LIN {X 0,Y 586.266,Z 608.093,A -85,B 0,C 180,E1 26221.406,E2 26221.406} C_VEL
LIN {X 0,Y 585.812,Z 650.287,A -85,B 0,C 180,E1 26218.326,E2 26218.326} C_VEL
LIN {X 0,Y 585.394,Z 696.233,A -85,B 0,C 180,E1 26215.061,E2 26215.061} C_VEL
LIN {X 0,Y 585.368,Z 709.809,A -85,B 0,C 180,E1 26214.141,E2 26214.141} C_VEL
LIN {X 0,Y 585.877,Z 715.244,A -85,B 0,C 180,E1 26214.043,E2 26214.043} C_VEL
LIN {X 0,Y 585.444,Z 927.531,A -85,B 0,C 180,E1 26211.27,E2 26211.27} C_VEL
LIN {X 0,Y 585.33,Z 946.86,A -85,B 0,C 180,E1 26210.828,E2 26210.828} C_VEL
LIN {X 0,Y 585.19,Z 964.794,A -85,B 0,C 180,E1 26210.242,E2 26210.242} C_VEL
LIN {X 0,Y 585.02,Z 982.786,A -85,B 0,C 180,E1 26209.467,E2 26209.467} C_VEL
LIN {X 0,Y 584.825,Z 1000.721,A -85,B 0,C 180,E1 26208.49,E2 26208.49} C_VEL
LIN {X 0,Y 584.635,Z 1017.158,A -85,B 0,C 180,E1 26207.388,E2 26207.388} C_VEL
LIN {X 0,Y 584.458,Z 1032.33,A -85,B 0,C 180,E1 26206.161,E2 26206.161} C_VEL
LIN {X 0,Y 584.295,Z 1046.685,A -85,B 0,C 180,E1 26204.772,E2 26204.772} C_VEL
LIN {X 0,Y 584.162,Z 1059.749,A -85,B 0,C 180,E1 26203.259,E2 26203.259} C_VEL
LIN {X 0,Y 584.061,Z 1071.294,A -85,B 0,C 180,E1 26201.654,E2 26201.654} C_VEL
LIN {X 0,Y 583.991,Z 1081.331,A -85,B 0,C 180,E1 26199.958,E2 26199.958} C_VEL
LIN {X 0,Y 583.953,Z 1089.534,A -85,B 0,C 180,E1 26198.244,E2 26198.244} C_VEL
LIN {X 0,Y 583.927,Z 1096.129,A -85,B 0,C 180,E1 26196.489,E2 26196.489} C_VEL
LIN {X 0,Y 583.916,Z 1101.299,A -85,B 0,C 180,E1 26194.616,E2 26194.616} C_VEL
LIN {X 0,Y 583.904,Z 1104.662,A -85,B 0,C 180,E1 26192.748,E2 26192.748} C_VEL
LIN {X 0,Y 583.911,Z 1106.306,A -85,B 0,C 180,E1 26190.883,E2 26190.883} C_VEL
LIN {X 0,Y 583.908,Z 1106.262,A -85,B 0,C 180,E1 26189.019,E2 26189.019} C_VEL
LIN {X 0,Y 583.906,Z 1104.537,A -85,B 0,C 180,E1 26187.153,E2 26187.153} C_VEL
LIN {X 0,Y 583.919,Z 1101.014,A -85,B 0,C 180,E1 26185.255,E2 26185.255} C_VEL
LIN {X 0,Y 583.926,Z 1095.819,A -85,B 0,C 180,E1 26183.412,E2 26183.412} C_VEL
LIN {X 0,Y 583.963,Z 1088.595,A -85,B 0,C 180,E1 26181.532,E2 26181.532} C_VEL
LIN {X 0,Y 584.009,Z 1079.736,A -85,B 0,C 180,E1 26179.743,E2 26179.743} C_VEL
LIN {X 0,Y 584.082,Z 1069.314,A -85,B 0,C 180,E1 26178.045,E2 26178.045} C_VEL
LIN {X 0,Y 584.186,Z 1057.326,A -85,B 0,C 180,E1 26176.439,E2 26176.439} C_VEL
LIN {X 0,Y 584.319,Z 1044.137,A -85,B 0,C 180,E1 26174.965,E2 26174.965} C_VEL
LIN {X 0,Y 584.478,Z 1029.579,A -85,B 0,C 180,E1 26173.604,E2 26173.604} C_VEL
LIN {X 0,Y 584.658,Z 1013.886,A -85,B 0,C 180,E1 26172.38,E2 26172.38} C_VEL
LIN {X 0,Y 584.848,Z 996.836,A -85,B 0,C 180,E1 26171.284,E2 26171.284} C_VEL
LIN {X 0,Y 585.039,Z 978.544,A -85,B 0,C 180,E1 26170.336,E2 26170.336} C_VEL
LIN {X 0,Y 585.211,Z 960.378,A -85,B 0,C 180,E1 26169.601,E2 26169.601} C_VEL
LIN {X 0,Y 585.358,Z 940.959,A -85,B 0,C 180,E1 26169.021,E2 26169.021} C_VEL
LIN {X 0,Y 585.468,Z 921.478,A -85,B 0,C 180,E1 26168.636,E2 26168.636} C_VEL
LIN {X 0,Y 585.728,Z 711.988,A -85,B 0,C 180,E1 26165.908,E2 26165.908} C_VEL
LIN {X 0,Y 585.285,Z 708.498,A -85,B 0,C 180,E1 26165.795,E2 26165.795} C_VEL
LIN {X 0,Y 585.682,Z 666.013,A -85,B 0,C 180,E1 26162.802,E2 26162.802} C_VEL
LIN {X 0,Y 586.142,Z 620.088,A -85,B 0,C 180,E1 26159.479,E2 26159.479} C_VEL
LIN {X 0,Y 586.104,Z 607.396,A -85,B 0,C 180,E1 26158.532,E2 26158.532} C_VEL
LIN {X 0,Y 584.094,Z 601.706,A -85,B 0,C 180,E1 26157.949,E2 26157.949} C_VEL
LIN {X 0,Y 584.092,Z 601.478,A -85,B 0,C 180,E1 26154.888,E2 26154.888} C_VEL
LIN {X 0,Y 584.068,Z 601.478,A -85,B 0,C 180,E1 26151.705,E2 26151.705} C_VEL
LIN {X 0,Y 584.088,Z 601.475,A -85,B 0,C 180,E1 26148.51,E2 26148.51} C_VEL
LIN {X 0,Y 584.079,Z 601.478,A -85,B 0,C 180,E1 26145.269,E2 26145.269} C_VEL
LIN {X 0,Y 584.092,Z 601.472,A -85,B 0,C 180,E1 26142.015,E2 26142.015} C_VEL
LIN {X 0,Y 584.093,Z 601.481,A -85,B 0,C 180,E1 26138.668,E2 26138.668} C_VEL
LIN {X 0,Y 584.089,Z 601.473,A -85,B 0,C 180,E1 26135.352,E2 26135.352} C_VEL
LIN {X 0,Y 584.073,Z 601.478,A -85,B 0,C 180,E1 26132.167,E2 26132.167} C_VEL
LIN {X 0,Y 584.091,Z 601.475,A -85,B 0,C 180,E1 26128.976,E2 26128.976} C_VEL
LIN {X 0,Y 584.063,Z 601.477,A -85,B 0,C 180,E1 26125.774,E2 26125.774} C_VEL
LIN {X 0,Y 584.096,Z 601.479,A -85,B 0,C 180,E1 26122.547,E2 26122.547} C_VEL
LIN {X 0,Y 584.058,Z 601.476,A -85,B 0,C 180,E1 26119.391,E2 26119.391} C_VEL
LIN {X 0,Y 584.09,Z 601.482,A -85,B 0,C 180,E1 26116.1,E2 26116.1} C_VEL
LIN {X 0,Y 584.06,Z 601.476,A -85,B 0,C 180,E1 26112.959,E2 26112.959} C_VEL
LIN {X 0,Y 584.053,Z 601.481,A -85,B 0,C 180,E1 26109.558,E2 26109.558} C_VEL
LIN {X 0,Y 584.073,Z 601.479,A -85,B 0,C 180,E1 26106.487,E2 26106.487} C_VEL
LIN {X 0,Y 584.084,Z 601.735,A -85,B 0,C 180,E1 26104.652,E2 26104.652} C_VEL
LIN {X 0,Y 584.958,Z 606.283,A -85,B 0,C 180,E1 26104.117,E2 26104.117} C_VEL
LIN {X 0,Y 584.765,Z 632.877,A -85,B 0,C 180,E1 26101.078,E2 26101.078} C_VEL
LIN {X 0,Y 584.541,Z 663.315,A -85,B 0,C 180,E1 26097.647,E2 26097.647} C_VEL
LIN {X 0,Y 584.373,Z 692.632,A -85,B 0,C 180,E1 26094.428,E2 26094.428} C_VEL
LIN {X 0,Y 584.842,Z 698.032,A -85,B 0,C 180,E1 26094.331,E2 26094.331} C_VEL
LIN {X 0,Y 584.731,Z 757.317,A -85,B 0,C 180,E1 26093.592,E2 26093.592} C_VEL
LIN {X 0,Y 583.768,Z 764.99,A -85,B 0,C 180,E1 26093.522,E2 26093.522} C_VEL
LIN {X 0,Y 577.692,Z 785.335,A -85,B 0,C 180,E1 26093.433,E2 26093.433} C_VEL
LIN {X 0,Y 576.962,Z 791.923,A -85,B 0,C 180,E1 26093.37,E2 26093.37} C_VEL
LIN {X 0,Y 576.9,Z 833.418,A -85,B 0,C 180,E1 26092.816,E2 26092.816} C_VEL
LIN {X 0,Y 576.808,Z 850.257,A -85,B 0,C 180,E1 26092.395,E2 26092.395} C_VEL
LIN {X 0,Y 576.673,Z 865.421,A -85,B 0,C 180,E1 26091.826,E2 26091.826} C_VEL
LIN {X 0,Y 576.524,Z 880.375,A -85,B 0,C 180,E1 26091.07,E2 26091.07} C_VEL
LIN {X 0,Y 576.387,Z 894.173,A -85,B 0,C 180,E1 26090.169,E2 26090.169} C_VEL
LIN {X 0,Y 576.244,Z 907.214,A -85,B 0,C 180,E1 26089.098,E2 26089.098} C_VEL
LIN {X 0,Y 576.128,Z 919.088,A -85,B 0,C 180,E1 26087.878,E2 26087.878} C_VEL
LIN {X 0,Y 576.036,Z 929.428,A -85,B 0,C 180,E1 26086.55,E2 26086.55} C_VEL
LIN {X 0,Y 575.976,Z 938.273,A -85,B 0,C 180,E1 26085.112,E2 26085.112} C_VEL
LIN {X 0,Y 575.94,Z 945.143,A -85,B 0,C 180,E1 26083.666,E2 26083.666} C_VEL
LIN {X 0,Y 575.921,Z 950.718,A -85,B 0,C 180,E1 26082.062,E2 26082.062} C_VEL
LIN {X 0,Y 575.916,Z 954.279,A -85,B 0,C 180,E1 26080.513,E2 26080.513} C_VEL
LIN {X 0,Y 575.913,Z 956.237,A -85,B 0,C 180,E1 26078.797,E2 26078.797} C_VEL
LIN {X 0,Y 575.915,Z 956.297,A -85,B 0,C 180,E1 26077.204,E2 26077.204} C_VEL
LIN {X 0,Y 575.916,Z 954.417,A -85,B 0,C 180,E1 26075.485,E2 26075.485} C_VEL
LIN {X 0,Y 575.921,Z 951.002,A -85,B 0,C 180,E1 26073.945,E2 26073.945} C_VEL
LIN {X 0,Y 575.937,Z 945.71,A -85,B 0,C 180,E1 26072.385,E2 26072.385} C_VEL
LIN {X 0,Y 575.972,Z 938.918,A -85,B 0,C 180,E1 26070.917,E2 26070.917} C_VEL
LIN {X 0,Y 576.033,Z 929.921,A -85,B 0,C 180,E1 26069.43,E2 26069.43} C_VEL
LIN {X 0,Y 576.127,Z 919.385,A -85,B 0,C 180,E1 26068.066,E2 26068.066} C_VEL
LIN {X 0,Y 576.239,Z 907.818,A -85,B 0,C 180,E1 26066.868,E2 26066.868} C_VEL
LIN {X 0,Y 576.376,Z 895.002,A -85,B 0,C 180,E1 26065.802,E2 26065.802} C_VEL
LIN {X 0,Y 576.518,Z 881.624,A -85,B 0,C 180,E1 26064.912,E2 26064.912} C_VEL
LIN {X 0,Y 576.662,Z 866.294,A -85,B 0,C 180,E1 26064.122,E2 26064.122} C_VEL
LIN {X 0,Y 576.807,Z 850.362,A -85,B 0,C 180,E1 26063.518,E2 26063.518} C_VEL
LIN {X 0,Y 576.897,Z 833.646,A -85,B 0,C 180,E1 26063.099,E2 26063.099} C_VEL
LIN {X 0,Y 576.958,Z 794.896,A -85,B 0,C 180,E1 26062.578,E2 26062.578} C_VEL
LIN {X 0,Y 576.936,Z 695.316,A -85,B 0,C 180,E1 26061.314,E2 26061.314} C_VEL
LIN {X 0,Y 576.519,Z 692.432,A -85,B 0,C 180,E1 26061.238,E2 26061.238} C_VEL
LIN {X 0,Y 576.769,Z 663.417,A -85,B 0,C 180,E1 26057.998,E2 26057.998} C_VEL
LIN {X 0,Y 577.081,Z 633.4,A -85,B 0,C 180,E1 26054.565,E2 26054.565} C_VEL
LIN {X 0,Y 577.283,Z 607.484,A -85,B 0,C 180,E1 26051.59,E2 26051.59} C_VEL
LIN {X 0,Y 576.093,Z 602.542,A -85,B 0,C 180,E1 26050.936,E2 26050.936} C_VEL
LIN {X 0,Y 576.161,Z 602.456,A -85,B 0,C 180,E1 26047.777,E2 26047.777} C_VEL
LIN {X 0,Y 576.088,Z 602.47,A -85,B 0,C 180,E1 26044.646,E2 26044.646} C_VEL
LIN {X 0,Y 576.163,Z 602.467,A -85,B 0,C 180,E1 26041.49,E2 26041.49} C_VEL
LIN {X 0,Y 576.094,Z 602.468,A -85,B 0,C 180,E1 26038.364,E2 26038.364} C_VEL
LIN {X 0,Y 576.159,Z 602.459,A -85,B 0,C 180,E1 26035.162,E2 26035.162} C_VEL
LIN {X 0,Y 576.1,Z 602.469,A -85,B 0,C 180,E1 26032.017,E2 26032.017} C_VEL
LIN {X 0,Y 576.154,Z 602.466,A -85,B 0,C 180,E1 26028.832,E2 26028.832} C_VEL
LIN {X 0,Y 576.106,Z 602.465,A -85,B 0,C 180,E1 26025.709,E2 26025.709} C_VEL
LIN {X 0,Y 576.145,Z 602.467,A -85,B 0,C 180,E1 26022.427,E2 26022.427} C_VEL
LIN {X 0,Y 576.16,Z 602.725,A -85,B 0,C 180,E1 26020.108,E2 26020.108} C_VEL
LIN {X 0,Y 577.539,Z 609.023,A -85,B 0,C 180,E1 26019.266,E2 26019.266} C_VEL
LIN {X 0,Y 577.051,Z 635.9,A -85,B 0,C 180,E1 26016.067,E2 26016.067} C_VEL
LIN {X 0,Y 576.75,Z 663.687,A -85,B 0,C 180,E1 26012.882,E2 26012.882} C_VEL
LIN {X 0,Y 576.515,Z 692.398,A -85,B 0,C 180,E1 26009.677,E2 26009.677} C_VEL
LIN {X 0,Y 577.137,Z 698.434,A -85,B 0,C 180,E1 26009.55,E2 26009.55} C_VEL
LIN {X 0,Y 576.9,Z 832.64,A -85,B 0,C 180,E1 26007.831,E2 26007.831} C_VEL
LIN {X 0,Y 576.81,Z 849.612,A -85,B 0,C 180,E1 26007.414,E2 26007.414} C_VEL
LIN {X 0,Y 576.689,Z 864.449,A -85,B 0,C 180,E1 26006.87,E2 26006.87} C_VEL
LIN {X 0,Y 576.537,Z 879.449,A -85,B 0,C 180,E1 26006.122,E2 26006.122} C_VEL
LIN {X 0,Y 576.396,Z 893.447,A -85,B 0,C 180,E1 26005.224,E2 26005.224} C_VEL
LIN {X 0,Y 576.254,Z 906.354,A -85,B 0,C 180,E1 26004.175,E2 26004.175} C_VEL
LIN {X 0,Y 576.139,Z 917.811,A -85,B 0,C 180,E1 26003.023,E2 26003.023} C_VEL
LIN {X 0,Y 576.047,Z 928.241,A -85,B 0,C 180,E1 26001.717,E2 26001.717} C_VEL
LIN {X 0,Y 575.98,Z 937.191,A -85,B 0,C 180,E1 26000.306,E2 26000.306} C_VEL
LIN {X 0,Y 575.944,Z 944.215,A -85,B 0,C 180,E1 25998.89,E2 25998.89} C_VEL
LIN {X 0,Y 575.926,Z 949.881,A -85,B 0,C 180,E1 25997.34,E2 25997.34} C_VEL
LIN {X 0,Y 575.916,Z 953.885,A -85,B 0,C 180,E1 25995.728,E2 25995.728} C_VEL
LIN {X 0,Y 575.914,Z 956.024,A -85,B 0,C 180,E1 25994.116,E2 25994.116} C_VEL
LIN {X 0,Y 575.915,Z 956.385,A -85,B 0,C 180,E1 25992.417,E2 25992.417} C_VEL
LIN {X 0,Y 575.917,Z 954.935,A -85,B 0,C 180,E1 25990.813,E2 25990.813} C_VEL
LIN {X 0,Y 575.923,Z 951.544,A -85,B 0,C 180,E1 25989.152,E2 25989.152} C_VEL
LIN {X 0,Y 575.936,Z 946.78,A -85,B 0,C 180,E1 25987.654,E2 25987.654} C_VEL
LIN {X 0,Y 575.963,Z 940.059,A -85,B 0,C 180,E1 25986.142,E2 25986.142} C_VEL
LIN {X 0,Y 576.021,Z 931.862,A -85,B 0,C 180,E1 25984.722,E2 25984.722} C_VEL
LIN {X 0,Y 576.098,Z 922.181,A -85,B 0,C 180,E1 25983.399,E2 25983.399} C_VEL
LIN {X 0,Y 576.214,Z 910.366,A -85,B 0,C 180,E1 25982.111,E2 25982.111} C_VEL
LIN {X 0,Y 576.342,Z 898.277,A -85,B 0,C 180,E1 25981.052,E2 25981.052} C_VEL
LIN {X 0,Y 576.483,Z 884.619,A -85,B 0,C 180,E1 25980.096,E2 25980.096} C_VEL
LIN {X 0,Y 576.628,Z 870.151,A -85,B 0,C 180,E1 25979.298,E2 25979.298} C_VEL
LIN {X 0,Y 576.765,Z 854.672,A -85,B 0,C 180,E1 25978.663,E2 25978.663} C_VEL
LIN {X 0,Y 576.881,Z 838.179,A -85,B 0,C 180,E1 25978.19,E2 25978.19} C_VEL
LIN {X 0,Y 576.944,Z 820.063,A -85,B 0,C 180,E1 25977.895,E2 25977.895} C_VEL
LIN {X 0,Y 576.927,Z 695.244,A -85,B 0,C 180,E1 25976.313,E2 25976.313} C_VEL
LIN {X 0,Y 576.533,Z 692.389,A -85,B 0,C 180,E1 25976.232,E2 25976.232} C_VEL
LIN {X 0,Y 576.751,Z 663.603,A -85,B 0,C 180,E1 25973.018,E2 25973.018} C_VEL
LIN {X 0,Y 577.106,Z 634.436,A -85,B 0,C 180,E1 25969.669,E2 25969.669} C_VEL
LIN {X 0,Y 577.548,Z 607.985,A -85,B 0,C 180,E1 25966.501,E2 25966.501} C_VEL
LIN {X 0,Y 576.165,Z 602.621,A -85,B 0,C 180,E1 25965.741,E2 25965.741} C_VEL
LIN {X 0,Y 576.144,Z 602.469,A -85,B 0,C 180,E1 25962.476,E2 25962.476} C_VEL
LIN {X 0,Y 576.14,Z 602.464,A -85,B 0,C 180,E1 25959.285,E2 25959.285} C_VEL
LIN {X 0,Y 576.142,Z 602.466,A -85,B 0,C 180,E1 25956.161,E2 25956.161} C_VEL
LIN {X 0,Y 576.142,Z 602.466,A -85,B 0,C 180,E1 25952.865,E2 25952.865} C_VEL
LIN {X 0,Y 576.143,Z 602.463,A -85,B 0,C 180,E1 25949.605,E2 25949.605} C_VEL
LIN {X 0,Y 576.156,Z 602.47,A -85,B 0,C 180,E1 25946.265,E2 25946.265} C_VEL
LIN {X 0,Y 576.152,Z 602.461,A -85,B 0,C 180,E1 25942.854,E2 25942.854} C_VEL
LIN {X 0,Y 576.14,Z 602.465,A -85,B 0,C 180,E1 25939.551,E2 25939.551} C_VEL
LIN {X 0,Y 576.145,Z 602.464,A -85,B 0,C 180,E1 25936.324,E2 25936.324} C_VEL
LIN {X 0,Y 576.136,Z 602.465,A -85,B 0,C 180,E1 25933.141,E2 25933.141} C_VEL
LIN {X 0,Y 576.146,Z 602.464,A -85,B 0,C 180,E1 25929.893,E2 25929.893} C_VEL
LIN {X 0,Y 576.137,Z 602.462,A -85,B 0,C 180,E1 25926.677,E2 25926.677} C_VEL
LIN {X 0,Y 576.156,Z 602.468,A -85,B 0,C 180,E1 25923.383,E2 25923.383} C_VEL
LIN {X 0,Y 576.156,Z 602.458,A -85,B 0,C 180,E1 25920,E2 25920} C_VEL
LIN {X 0,Y 576.139,Z 602.465,A -85,B 0,C 180,E1 25916.717,E2 25916.717} C_VEL
LIN {X 0,Y 576.151,Z 602.462,A -85,B 0,C 180,E1 25913.423,E2 25913.423} C_VEL
LIN {X 0,Y 576.132,Z 602.464,A -85,B 0,C 180,E1 25910.208,E2 25910.208} C_VEL
LIN {X 0,Y 576.15,Z 602.465,A -85,B 0,C 180,E1 25906.962,E2 25906.962} C_VEL
LIN {X 0,Y 576.13,Z 602.464,A -85,B 0,C 180,E1 25903.775,E2 25903.775} C_VEL
LIN {X 0,Y 576.153,Z 602.465,A -85,B 0,C 180,E1 25900.537,E2 25900.537} C_VEL
LIN {X 0,Y 576.142,Z 602.46,A -85,B 0,C 180,E1 25897.232,E2 25897.232} C_VEL
LIN {X 0,Y 576.139,Z 602.467,A -85,B 0,C 180,E1 25893.795,E2 25893.795} C_VEL
LIN {X 0,Y 576.159,Z 602.461,A -85,B 0,C 180,E1 25890.586,E2 25890.586} C_VEL
LIN {X 0,Y 576.128,Z 602.467,A -85,B 0,C 180,E1 25887.321,E2 25887.321} C_VEL
LIN {X 0,Y 576.153,Z 602.463,A -85,B 0,C 180,E1 25884.086,E2 25884.086} C_VEL
LIN {X 0,Y 576.125,Z 602.466,A -85,B 0,C 180,E1 25880.874,E2 25880.874} C_VEL
LIN {X 0,Y 576.155,Z 602.467,A -85,B 0,C 180,E1 25877.67,E2 25877.67} C_VEL
LIN {X 0,Y 576.125,Z 602.465,A -85,B 0,C 180,E1 25874.497,E2 25874.497} C_VEL
LIN {X 0,Y 576.158,Z 602.468,A -85,B 0,C 180,E1 25871.258,E2 25871.258} C_VEL
LIN {X 0,Y 576.132,Z 602.464,A -85,B 0,C 180,E1 25868.01,E2 25868.01} C_VEL
LIN {X 0,Y 576.135,Z 602.466,A -85,B 0,C 180,E1 25864.576,E2 25864.576} C_VEL
LIN {X 0,Y 576.158,Z 602.644,A -85,B 0,C 180,E1 25862.486,E2 25862.486} C_VEL
LIN {X 0,Y 578.333,Z 608.935,A -85,B 0,C 180,E1 25861.823,E2 25861.823} C_VEL
LIN {X 0,Y 579.059,Z 611.232,A -85,B 0,C 180,E1 25861.604,E2 25861.604} C_VEL
LIN {X 0,Y 578.46,Z 654.116,A -85,B 0,C 180,E1 25858.437,E2 25858.437} C_VEL
LIN {X 0,Y 577.882,Z 700.062,A -85,B 0,C 180,E1 25855.136,E2 25855.136} C_VEL
LIN {X 0,Y 577.877,Z 709.884,A -85,B 0,C 180,E1 25854.473,E2 25854.473} C_VEL
LIN {X 0,Y 578.569,Z 715.892,A -85,B 0,C 180,E1 25854.358,E2 25854.358} C_VEL
LIN {X 0,Y 577.986,Z 927.53,A -85,B 0,C 180,E1 25851.558,E2 25851.558} C_VEL
LIN {X 0,Y 577.831,Z 946.932,A -85,B 0,C 180,E1 25851.109,E2 25851.109} C_VEL
LIN {X 0,Y 577.643,Z 964.794,A -85,B 0,C 180,E1 25850.519,E2 25850.519} C_VEL
LIN {X 0,Y 577.411,Z 982.787,A -85,B 0,C 180,E1 25849.735,E2 25849.735} C_VEL
LIN {X 0,Y 577.152,Z 1000.542,A -85,B 0,C 180,E1 25848.756,E2 25848.756} C_VEL
LIN {X 0,Y 576.898,Z 1016.794,A -85,B 0,C 180,E1 25847.656,E2 25847.656} C_VEL
LIN {X 0,Y 576.649,Z 1032.553,A -85,B 0,C 180,E1 25846.365,E2 25846.365} C_VEL
LIN {X 0,Y 576.432,Z 1046.938,A -85,B 0,C 180,E1 25844.95,E2 25844.95} C_VEL
LIN {X 0,Y 576.258,Z 1059.75,A -85,B 0,C 180,E1 25843.444,E2 25843.444} C_VEL
LIN {X 0,Y 576.117,Z 1071.332,A -85,B 0,C 180,E1 25841.811,E2 25841.811} C_VEL
LIN {X 0,Y 576.028,Z 1081.332,A -85,B 0,C 180,E1 25840.097,E2 25840.097} C_VEL
LIN {X 0,Y 575.967,Z 1089.732,A -85,B 0,C 180,E1 25838.31,E2 25838.31} C_VEL
LIN {X 0,Y 575.932,Z 1096.432,A -85,B 0,C 180,E1 25836.479,E2 25836.479} C_VEL
LIN {X 0,Y 575.918,Z 1101.298,A -85,B 0,C 180,E1 25834.68,E2 25834.68} C_VEL
LIN {X 0,Y 575.905,Z 1104.661,A -85,B 0,C 180,E1 25832.786,E2 25832.786} C_VEL
LIN {X 0,Y 575.911,Z 1106.305,A -85,B 0,C 180,E1 25830.895,E2 25830.895} C_VEL
LIN {X 0,Y 575.908,Z 1106.263,A -85,B 0,C 180,E1 25829.005,E2 25829.005} C_VEL
LIN {X 0,Y 575.907,Z 1104.537,A -85,B 0,C 180,E1 25827.114,E2 25827.114} C_VEL
LIN {X 0,Y 575.92,Z 1101.086,A -85,B 0,C 180,E1 25825.22,E2 25825.22} C_VEL
LIN {X 0,Y 575.931,Z 1095.819,A -85,B 0,C 180,E1 25823.32,E2 25823.32} C_VEL
LIN {X 0,Y 575.98,Z 1088.594,A -85,B 0,C 180,E1 25821.414,E2 25821.414} C_VEL
LIN {X 0,Y 576.044,Z 1079.736,A -85,B 0,C 180,E1 25819.6,E2 25819.6} C_VEL
LIN {X 0,Y 576.146,Z 1069.313,A -85,B 0,C 180,E1 25817.878,E2 25817.878} C_VEL
LIN {X 0,Y 576.285,Z 1057.325,A -85,B 0,C 180,E1 25816.249,E2 25816.249} C_VEL
LIN {X 0,Y 576.463,Z 1044.233,A -85,B 0,C 180,E1 25814.765,E2 25814.765} C_VEL
LIN {X 0,Y 576.681,Z 1029.581,A -85,B 0,C 180,E1 25813.376,E2 25813.376} C_VEL
LIN {X 0,Y 576.925,Z 1013.888,A -85,B 0,C 180,E1 25812.136,E2 25812.136} C_VEL
LIN {X 0,Y 577.175,Z 997.405,A -85,B 0,C 180,E1 25811.059,E2 25811.059} C_VEL
LIN {X 0,Y 577.43,Z 979.798,A -85,B 0,C 180,E1 25810.125,E2 25810.125} C_VEL
LIN {X 0,Y 577.663,Z 961.495,A -85,B 0,C 180,E1 25809.363,E2 25809.363} C_VEL
LIN {X 0,Y 577.861,Z 942.593,A -85,B 0,C 180,E1 25808.777,E2 25808.777} C_VEL
LIN {X 0,Y 578.008,Z 923.513,A -85,B 0,C 180,E1 25808.378,E2 25808.378} C_VEL
LIN {X 0,Y 578.407,Z 713.038,A -85,B 0,C 180,E1 25805.597,E2 25805.597} C_VEL
LIN {X 0,Y 577.796,Z 708.995,A -85,B 0,C 180,E1 25805.491,E2 25805.491} C_VEL
LIN {X 0,Y 578.321,Z 666.436,A -85,B 0,C 180,E1 25802.458,E2 25802.458} C_VEL
LIN {X 0,Y 578.921,Z 621.115,A -85,B 0,C 180,E1 25799.134,E2 25799.134} C_VEL
LIN {X 0,Y 578.877,Z 610.459,A -85,B 0,C 180,E1 25798.326,E2 25798.326} C_VEL
LIN {X 0,Y 576.164,Z 602.67,A -85,B 0,C 180,E1 25797.524,E2 25797.524} C_VEL
LIN {X 0,Y 576.144,Z 602.464,A -85,B 0,C 180,E1 25794.208,E2 25794.208} C_VEL
LIN {X 0,Y 576.157,Z 602.47,A -85,B 0,C 180,E1 25790.953,E2 25790.953} C_VEL
LIN {X 0,Y 576.136,Z 602.464,A -85,B 0,C 180,E1 25787.672,E2 25787.672} C_VEL
LIN {X 0,Y 576.144,Z 602.465,A -85,B 0,C 180,E1 25784.498,E2 25784.498} C_VEL
LIN {X 0,Y 576.141,Z 602.466,A -85,B 0,C 180,E1 25781.259,E2 25781.259} C_VEL
LIN {X 0,Y 576.142,Z 602.463,A -85,B 0,C 180,E1 25778.011,E2 25778.011} C_VEL
LIN {X 0,Y 576.157,Z 602.47,A -85,B 0,C 180,E1 25774.656,E2 25774.656} C_VEL
LIN {X 0,Y 576.156,Z 602.462,A -85,B 0,C 180,E1 25771.257,E2 25771.257} C_VEL
LIN {X 0,Y 576.131,Z 602.467,A -85,B 0,C 180,E1 25768.054,E2 25768.054} C_VEL
LIN {X 0,Y 576.155,Z 602.465,A -85,B 0,C 180,E1 25764.821,E2 25764.821} C_VEL
LIN {X 0,Y 576.12,Z 602.466,A -85,B 0,C 180,E1 25761.588,E2 25761.588} C_VEL
LIN {X 0,Y 576.16,Z 602.47,A -85,B 0,C 180,E1 25758.307,E2 25758.307} C_VEL
LIN {X 0,Y 576.12,Z 602.466,A -85,B 0,C 180,E1 25755.089,E2 25755.089} C_VEL
LIN {X 0,Y 576.123,Z 602.471,A -85,B 0,C 180,E1 25751.715,E2 25751.715} C_VEL
LIN {X 0,Y 576.135,Z 602.466,A -85,B 0,C 180,E1 25748.583,E2 25748.583} C_VEL
LIN {X 0,Y 576.106,Z 602.475,A -85,B 0,C 180,E1 25745.377,E2 25745.377} C_VEL
LIN {X 0,Y 576.134,Z 602.717,A -85,B 0,C 180,E1 25744.853,E2 25744.853} C_VEL
LIN {X 0,Y 577.251,Z 608.642,A -85,B 0,C 180,E1 25744.172,E2 25744.172} C_VEL
LIN {X 0,Y 577.025,Z 637.299,A -85,B 0,C 180,E1 25740.893,E2 25740.893} C_VEL
LIN {X 0,Y 576.742,Z 666.044,A -85,B 0,C 180,E1 25737.615,E2 25737.615} C_VEL
LIN {X 0,Y 576.545,Z 692.765,A -85,B 0,C 180,E1 25734.651,E2 25734.651} C_VEL
LIN {X 0,Y 577.165,Z 698.813,A -85,B 0,C 180,E1 25734.545,E2 25734.545} C_VEL
LIN {X 0,Y 576.962,Z 791.923,A -85,B 0,C 180,E1 25733.37,E2 25733.37} C_VEL
LIN {X 0,Y 575.998,Z 799.601,A -85,B 0,C 180,E1 25733.302,E2 25733.302} C_VEL
LIN {X 0,Y 569.926,Z 819.95,A -85,B 0,C 180,E1 25733.213,E2 25733.213} C_VEL
LIN {X 0,Y 569.189,Z 826.523,A -85,B 0,C 180,E1 25733.137,E2 25733.137} C_VEL
LIN {X 0,Y 569.102,Z 843.512,A -85,B 0,C 180,E1 25732.793,E2 25732.793} C_VEL
LIN {X 0,Y 568.951,Z 859.326,A -85,B 0,C 180,E1 25732.274,E2 25732.274} C_VEL
LIN {X 0,Y 568.758,Z 874.934,A -85,B 0,C 180,E1 25731.559,E2 25731.559} C_VEL
LIN {X 0,Y 568.57,Z 889.287,A -85,B 0,C 180,E1 25730.689,E2 25730.689} C_VEL
LIN {X 0,Y 568.4,Z 902.656,A -85,B 0,C 180,E1 25729.663,E2 25729.663} C_VEL
LIN {X 0,Y 568.244,Z 914.474,A -85,B 0,C 180,E1 25728.531,E2 25728.531} C_VEL
LIN {X 0,Y 568.117,Z 924.963,A -85,B 0,C 180,E1 25727.291,E2 25727.291} C_VEL
LIN {X 0,Y 568.024,Z 934.338,A -85,B 0,C 180,E1 25725.906,E2 25725.906} C_VEL
LIN {X 0,Y 567.968,Z 941.956,A -85,B 0,C 180,E1 25724.479,E2 25724.479} C_VEL
LIN {X 0,Y 567.93,Z 948.286,A -85,B 0,C 180,E1 25722.902,E2 25722.902} C_VEL
LIN {X 0,Y 567.92,Z 952.814,A -85,B 0,C 180,E1 25721.296,E2 25721.296} C_VEL
LIN {X 0,Y 567.915,Z 955.468,A -85,B 0,C 180,E1 25719.706,E2 25719.706} C_VEL
LIN {X 0,Y 567.919,Z 956.499,A -85,B 0,C 180,E1 25717.975,E2 25717.975} C_VEL
LIN {X 0,Y 567.915,Z 955.548,A -85,B 0,C 180,E1 25716.278,E2 25716.278} C_VEL
LIN {X 0,Y 567.917,Z 952.935,A -85,B 0,C 180,E1 25714.671,E2 25714.671} C_VEL
LIN {X 0,Y 567.931,Z 948.589,A -85,B 0,C 180,E1 25713.098,E2 25713.098} C_VEL
LIN {X 0,Y 567.963,Z 942.292,A -85,B 0,C 180,E1 25711.505,E2 25711.505} C_VEL
LIN {X 0,Y 568.025,Z 934.327,A -85,B 0,C 180,E1 25710.002,E2 25710.002} C_VEL
LIN {X 0,Y 568.121,Z 924.841,A -85,B 0,C 180,E1 25708.603,E2 25708.603} C_VEL
LIN {X 0,Y 568.251,Z 913.769,A -85,B 0,C 180,E1 25707.304,E2 25707.304} C_VEL
LIN {X 0,Y 568.423,Z 901.227,A -85,B 0,C 180,E1 25706.125,E2 25706.125} C_VEL
LIN {X 0,Y 568.602,Z 886.939,A -85,B 0,C 180,E1 25705.062,E2 25705.062} C_VEL
LIN {X 0,Y 568.789,Z 872.321,A -85,B 0,C 180,E1 25704.217,E2 25704.217} C_VEL
LIN {X 0,Y 568.977,Z 857.409,A -85,B 0,C 180,E1 25703.561,E2 25703.561} C_VEL
LIN {X 0,Y 569.11,Z 841.392,A -85,B 0,C 180,E1 25703.064,E2 25703.064} C_VEL
LIN {X 0,Y 569.199,Z 824.674,A -85,B 0,C 180,E1 25702.745,E2 25702.745} C_VEL
LIN {X 0,Y 569.272,Z 696.268,A -85,B 0,C 180,E1 25701.095,E2 25701.095} C_VEL
LIN {X 0,Y 568.688,Z 692.321,A -85,B 0,C 180,E1 25700.991,E2 25700.991} C_VEL
LIN {X 0,Y 569.013,Z 662.912,A -85,B 0,C 180,E1 25697.656,E2 25697.656} C_VEL
LIN {X 0,Y 569.398,Z 634.334,A -85,B 0,C 180,E1 25694.338,E2 25694.338} C_VEL
LIN {X 0,Y 569.589,Z 609.635,A -85,B 0,C 180,E1 25691.504,E2 25691.504} C_VEL
LIN {X 0,Y 568.162,Z 603.569,A -85,B 0,C 180,E1 25690.71,E2 25690.71} C_VEL
LIN {X 0,Y 568.192,Z 603.446,A -85,B 0,C 180,E1 25687.473,E2 25687.473} C_VEL
LIN {X 0,Y 568.152,Z 603.46,A -85,B 0,C 180,E1 25684.519,E2 25684.519} C_VEL
LIN {X 0,Y 568.204,Z 603.455,A -85,B 0,C 180,E1 25681.273,E2 25681.273} C_VEL
LIN {X 0,Y 568.157,Z 603.457,A -85,B 0,C 180,E1 25678.255,E2 25678.255} C_VEL
LIN {X 0,Y 568.203,Z 603.447,A -85,B 0,C 180,E1 25674.982,E2 25674.982} C_VEL
LIN {X 0,Y 568.166,Z 603.458,A -85,B 0,C 180,E1 25671.906,E2 25671.906} C_VEL
LIN {X 0,Y 568.191,Z 603.455,A -85,B 0,C 180,E1 25668.573,E2 25668.573} C_VEL
LIN {X 0,Y 568.185,Z 603.454,A -85,B 0,C 180,E1 25665.41,E2 25665.41} C_VEL
LIN {X 0,Y 568.177,Z 603.46,A -85,B 0,C 180,E1 25662.088,E2 25662.088} C_VEL
LIN {X 0,Y 568.249,Z 603.694,A -85,B 0,C 180,E1 25660.442,E2 25660.442} C_VEL
LIN {X 0,Y 569.982,Z 611.432,A -85,B 0,C 180,E1 25659.389,E2 25659.389} C_VEL
LIN {X 0,Y 569.439,Z 637.562,A -85,B 0,C 180,E1 25656.25,E2 25656.25} C_VEL
LIN {X 0,Y 568.971,Z 664.938,A -85,B 0,C 180,E1 25653.022,E2 25653.022} C_VEL
LIN {X 0,Y 568.701,Z 692.615,A -85,B 0,C 180,E1 25649.9,E2 25649.9} C_VEL
LIN {X 0,Y 569.469,Z 699.435,A -85,B 0,C 180,E1 25649.768,E2 25649.768} C_VEL
LIN {X 0,Y 569.165,Z 832.659,A -85,B 0,C 180,E1 25648.037,E2 25648.037} C_VEL
LIN {X 0,Y 569.05,Z 849.638,A -85,B 0,C 180,E1 25647.615,E2 25647.615} C_VEL
LIN {X 0,Y 568.903,Z 864.121,A -85,B 0,C 180,E1 25647.079,E2 25647.079} C_VEL
LIN {X 0,Y 568.712,Z 879.194,A -85,B 0,C 180,E1 25646.321,E2 25646.321} C_VEL
LIN {X 0,Y 568.524,Z 893.256,A -85,B 0,C 180,E1 25645.411,E2 25645.411} C_VEL
LIN {X 0,Y 568.352,Z 906.201,A -85,B 0,C 180,E1 25644.347,E2 25644.347} C_VEL
LIN {X 0,Y 568.2,Z 918.146,A -85,B 0,C 180,E1 25643.128,E2 25643.128} C_VEL
LIN {X 0,Y 568.082,Z 928.497,A -85,B 0,C 180,E1 25641.804,E2 25641.804} C_VEL
LIN {X 0,Y 567.997,Z 937.652,A -85,B 0,C 180,E1 25640.329,E2 25640.329} C_VEL
LIN {X 0,Y 567.949,Z 944.776,A -85,B 0,C 180,E1 25638.834,E2 25638.834} C_VEL
LIN {X 0,Y 567.926,Z 950.533,A -85,B 0,C 180,E1 25637.184,E2 25637.184} C_VEL
LIN {X 0,Y 567.921,Z 954.149,A -85,B 0,C 180,E1 25635.627,E2 25635.627} C_VEL
LIN {X 0,Y 567.914,Z 956.144,A -85,B 0,C 180,E1 25633.954,E2 25633.954} C_VEL
LIN {X 0,Y 567.914,Z 956.344,A -85,B 0,C 180,E1 25632.266,E2 25632.266} C_VEL
LIN {X 0,Y 567.915,Z 954.595,A -85,B 0,C 180,E1 25630.565,E2 25630.565} C_VEL
LIN {X 0,Y 567.927,Z 951.1,A -85,B 0,C 180,E1 25628.922,E2 25628.922} C_VEL
LIN {X 0,Y 567.944,Z 945.762,A -85,B 0,C 180,E1 25627.323,E2 25627.323} C_VEL
LIN {X 0,Y 567.992,Z 938.631,A -85,B 0,C 180,E1 25625.764,E2 25625.764} C_VEL
LIN {X 0,Y 568.065,Z 929.929,A -85,B 0,C 180,E1 25624.314,E2 25624.314} C_VEL
LIN {X 0,Y 568.185,Z 919.399,A -85,B 0,C 180,E1 25622.928,E2 25622.928} C_VEL
LIN {X 0,Y 568.323,Z 908.264,A -85,B 0,C 180,E1 25621.754,E2 25621.754} C_VEL
LIN {X 0,Y 568.507,Z 894.779,A -85,B 0,C 180,E1 25620.614,E2 25620.614} C_VEL
LIN {X 0,Y 568.691,Z 880.877,A -85,B 0,C 180,E1 25619.686,E2 25619.686} C_VEL
LIN {X 0,Y 568.881,Z 865.353,A -85,B 0,C 180,E1 25618.887,E2 25618.887} C_VEL
LIN {X 0,Y 569.048,Z 849.908,A -85,B 0,C 180,E1 25618.303,E2 25618.303} C_VEL
LIN {X 0,Y 569.166,Z 832.986,A -85,B 0,C 180,E1 25617.879,E2 25617.879} C_VEL
LIN {X 0,Y 569.347,Z 754.576,A -85,B 0,C 180,E1 25616.849,E2 25616.849} C_VEL
LIN {X 0,Y 569.244,Z 696.076,A -85,B 0,C 180,E1 25616.092,E2 25616.092} C_VEL
LIN {X 0,Y 568.716,Z 692.567,A -85,B 0,C 180,E1 25616.008,E2 25616.008} C_VEL
LIN {X 0,Y 568.976,Z 664.232,A -85,B 0,C 180,E1 25612.807,E2 25612.807} C_VEL
LIN {X 0,Y 569.513,Z 635.665,A -85,B 0,C 180,E1 25609.43,E2 25609.43} C_VEL
LIN {X 0,Y 570.03,Z 610.535,A -85,B 0,C 180,E1 25606.385,E2 25606.385} C_VEL
LIN {X 0,Y 568.213,Z 603.539,A -85,B 0,C 180,E1 25605.373,E2 25605.373} C_VEL
LIN {X 0,Y 568.213,Z 603.454,A -85,B 0,C 180,E1 25602.049,E2 25602.049} C_VEL
LIN {X 0,Y 568.216,Z 603.458,A -85,B 0,C 180,E1 25598.622,E2 25598.622} C_VEL
LIN {X 0,Y 568.206,Z 603.453,A -85,B 0,C 180,E1 25595.252,E2 25595.252} C_VEL
LIN {X 0,Y 568.202,Z 603.453,A -85,B 0,C 180,E1 25591.983,E2 25591.983} C_VEL
LIN {X 0,Y 568.204,Z 603.455,A -85,B 0,C 180,E1 25588.711,E2 25588.711} C_VEL
LIN {X 0,Y 568.205,Z 603.45,A -85,B 0,C 180,E1 25585.427,E2 25585.427} C_VEL
LIN {X 0,Y 568.222,Z 603.456,A -85,B 0,C 180,E1 25582.012,E2 25582.012} C_VEL
LIN {X 0,Y 568.213,Z 603.448,A -85,B 0,C 180,E1 25578.679,E2 25578.679} C_VEL
LIN {X 0,Y 568.199,Z 603.453,A -85,B 0,C 180,E1 25575.353,E2 25575.353} C_VEL
LIN {X 0,Y 568.206,Z 603.454,A -85,B 0,C 180,E1 25572.088,E2 25572.088} C_VEL
LIN {X 0,Y 568.199,Z 603.452,A -85,B 0,C 180,E1 25568.806,E2 25568.806} C_VEL
LIN {X 0,Y 568.216,Z 603.455,A -85,B 0,C 180,E1 25565.453,E2 25565.453} C_VEL
LIN {X 0,Y 568.216,Z 603.449,A -85,B 0,C 180,E1 25562.017,E2 25562.017} C_VEL
LIN {X 0,Y 568.198,Z 603.456,A -85,B 0,C 180,E1 25558.689,E2 25558.689} C_VEL
LIN {X 0,Y 568.209,Z 603.449,A -85,B 0,C 180,E1 25555.458,E2 25555.458} C_VEL
LIN {X 0,Y 568.194,Z 603.451,A -85,B 0,C 180,E1 25552.187,E2 25552.187} C_VEL
LIN {X 0,Y 568.212,Z 603.454,A -85,B 0,C 180,E1 25548.942,E2 25548.942} C_VEL
LIN {X 0,Y 568.201,Z 603.448,A -85,B 0,C 180,E1 25545.634,E2 25545.634} C_VEL
LIN {X 0,Y 568.211,Z 603.455,A -85,B 0,C 180,E1 25542.277,E2 25542.277} C_VEL
LIN {X 0,Y 568.219,Z 603.45,A -85,B 0,C 180,E1 25538.963,E2 25538.963} C_VEL
LIN {X 0,Y 568.192,Z 603.456,A -85,B 0,C 180,E1 25535.684,E2 25535.684} C_VEL
LIN {X 0,Y 568.212,Z 603.451,A -85,B 0,C 180,E1 25532.433,E2 25532.433} C_VEL
LIN {X 0,Y 568.188,Z 603.451,A -85,B 0,C 180,E1 25529.176,E2 25529.176} C_VEL
LIN {X 0,Y 568.218,Z 603.459,A -85,B 0,C 180,E1 25525.853,E2 25525.853} C_VEL
LIN {X 0,Y 568.208,Z 603.45,A -85,B 0,C 180,E1 25522.494,E2 25522.494} C_VEL
LIN {X 0,Y 568.194,Z 603.457,A -85,B 0,C 180,E1 25519.11,E2 25519.11} C_VEL
LIN {X 0,Y 568.216,Z 603.451,A -85,B 0,C 180,E1 25515.828,E2 25515.828} C_VEL
LIN {X 0,Y 568.185,Z 603.456,A -85,B 0,C 180,E1 25512.645,E2 25512.645} C_VEL
LIN {X 0,Y 568.214,Z 603.455,A -85,B 0,C 180,E1 25509.422,E2 25509.422} C_VEL
LIN {X 0,Y 568.183,Z 603.459,A -85,B 0,C 180,E1 25506.247,E2 25506.247} C_VEL
LIN {X 0,Y 568.236,Z 603.576,A -85,B 0,C 180,E1 25502.936,E2 25502.936} C_VEL
LIN {X 0,Y 569.117,Z 606.324,A -85,B 0,C 180,E1 25502.604,E2 25502.604} C_VEL
LIN {X 0,Y 571.861,Z 614.244,A -85,B 0,C 180,E1 25501.817,E2 25501.817} C_VEL
LIN {X 0,Y 571.118,Z 657.179,A -85,B 0,C 180,E1 25498.608,E2 25498.608} C_VEL
LIN {X 0,Y 570.397,Z 702.359,A -85,B 0,C 180,E1 25495.322,E2 25495.322} C_VEL
LIN {X 0,Y 570.403,Z 709.925,A -85,B 0,C 180,E1 25494.814,E2 25494.814} C_VEL
LIN {X 0,Y 571.278,Z 716.949,A -85,B 0,C 180,E1 25494.675,E2 25494.675} C_VEL
LIN {X 0,Y 570.542,Z 927.53,A -85,B 0,C 180,E1 25491.853,E2 25491.853} C_VEL
LIN {X 0,Y 570.347,Z 946.916,A -85,B 0,C 180,E1 25491.4,E2 25491.4} C_VEL
LIN {X 0,Y 570.097,Z 965.379,A -85,B 0,C 180,E1 25490.779,E2 25490.779} C_VEL
LIN {X 0,Y 569.797,Z 983.66,A -85,B 0,C 180,E1 25489.964,E2 25489.964} C_VEL
LIN {X 0,Y 569.476,Z 1001.046,A -85,B 0,C 180,E1 25488.986,E2 25488.986} C_VEL
LIN {X 0,Y 569.151,Z 1017.469,A -85,B 0,C 180,E1 25487.851,E2 25487.851} C_VEL
LIN {X 0,Y 568.841,Z 1033.107,A -85,B 0,C 180,E1 25486.544,E2 25486.544} C_VEL
LIN {X 0,Y 568.568,Z 1047.432,A -85,B 0,C 180,E1 25485.106,E2 25485.106} C_VEL
LIN {X 0,Y 568.342,Z 1060.525,A -85,B 0,C 180,E1 25483.531,E2 25483.531} C_VEL
LIN {X 0,Y 568.169,Z 1071.934,A -85,B 0,C 180,E1 25481.882,E2 25481.882} C_VEL
LIN {X 0,Y 568.055,Z 1081.85,A -85,B 0,C 180,E1 25480.137,E2 25480.137} C_VEL
LIN {X 0,Y 567.978,Z 1090.244,A -85,B 0,C 180,E1 25478.299,E2 25478.299} C_VEL
LIN {X 0,Y 567.937,Z 1096.735,A -85,B 0,C 180,E1 25476.469,E2 25476.469} C_VEL
LIN {X 0,Y 567.918,Z 1101.504,A -85,B 0,C 180,E1 25474.645,E2 25474.645} C_VEL
LIN {X 0,Y 567.905,Z 1104.775,A -85,B 0,C 180,E1 25472.724,E2 25472.724} C_VEL
LIN {X 0,Y 567.912,Z 1106.328,A -85,B 0,C 180,E1 25470.807,E2 25470.807} C_VEL
LIN {X 0,Y 567.905,Z 1106.197,A -85,B 0,C 180,E1 25468.89,E2 25468.89} C_VEL
LIN {X 0,Y 567.911,Z 1104.383,A -85,B 0,C 180,E1 25466.972,E2 25466.972} C_VEL
LIN {X 0,Y 567.919,Z 1100.842,A -85,B 0,C 180,E1 25465.051,E2 25465.051} C_VEL
LIN {X 0,Y 567.939,Z 1095.475,A -85,B 0,C 180,E1 25463.124,E2 25463.124} C_VEL
LIN {X 0,Y 567.995,Z 1088.594,A -85,B 0,C 180,E1 25461.292,E2 25461.292} C_VEL
LIN {X 0,Y 568.081,Z 1079.735,A -85,B 0,C 180,E1 25459.452,E2 25459.452} C_VEL
LIN {X 0,Y 568.209,Z 1069.312,A -85,B 0,C 180,E1 25457.706,E2 25457.706} C_VEL
LIN {X 0,Y 568.391,Z 1057.325,A -85,B 0,C 180,E1 25456.054,E2 25456.054} C_VEL
LIN {X 0,Y 568.619,Z 1044.233,A -85,B 0,C 180,E1 25454.55,E2 25454.55} C_VEL
LIN {X 0,Y 568.899,Z 1029.583,A -85,B 0,C 180,E1 25453.142,E2 25453.142} C_VEL
LIN {X 0,Y 569.216,Z 1013.532,A -85,B 0,C 180,E1 25451.859,E2 25451.859} C_VEL
LIN {X 0,Y 569.541,Z 996.289,A -85,B 0,C 180,E1 25450.728,E2 25450.728} C_VEL
LIN {X 0,Y 569.866,Z 978.304,A -85,B 0,C 180,E1 25449.778,E2 25449.778} C_VEL
LIN {X 0,Y 570.156,Z 959.647,A -85,B 0,C 180,E1 25449.011,E2 25449.011} C_VEL
LIN {X 0,Y 570.397,Z 940.355,A -85,B 0,C 180,E1 25448.427,E2 25448.427} C_VEL
LIN {X 0,Y 570.578,Z 921.05,A -85,B 0,C 180,E1 25448.043,E2 25448.043} C_VEL
LIN {X 0,Y 571.12,Z 714.226,A -85,B 0,C 180,E1 25445.281,E2 25445.281} C_VEL
LIN {X 0,Y 570.338,Z 709.304,A -85,B 0,C 180,E1 25445.163,E2 25445.163} C_VEL
LIN {X 0,Y 570.96,Z 667.78,A -85,B 0,C 180,E1 25442.172,E2 25442.172} C_VEL
LIN {X 0,Y 571.711,Z 622.711,A -85,B 0,C 180,E1 25438.823,E2 25438.823} C_VEL
LIN {X 0,Y 571.695,Z 613.522,A -85,B 0,C 180,E1 25438.117,E2 25438.117} C_VEL
LIN {X 0,Y 568.249,Z 603.672,A -85,B 0,C 180,E1 25437.094,E2 25437.094} C_VEL
LIN {X 0,Y 568.191,Z 603.456,A -85,B 0,C 180,E1 25433.873,E2 25433.873} C_VEL
LIN {X 0,Y 568.211,Z 603.456,A -85,B 0,C 180,E1 25430.692,E2 25430.692} C_VEL
LIN {X 0,Y 568.196,Z 603.455,A -85,B 0,C 180,E1 25427.489,E2 25427.489} C_VEL
LIN {X 0,Y 568.213,Z 603.45,A -85,B 0,C 180,E1 25424.173,E2 25424.173} C_VEL
LIN {X 0,Y 568.219,Z 603.459,A -85,B 0,C 180,E1 25420.755,E2 25420.755} C_VEL
LIN {X 0,Y 568.209,Z 603.452,A -85,B 0,C 180,E1 25417.379,E2 25417.379} C_VEL
LIN {X 0,Y 568.197,Z 603.455,A -85,B 0,C 180,E1 25414.149,E2 25414.149} C_VEL
LIN {X 0,Y 568.213,Z 603.456,A -85,B 0,C 180,E1 25410.827,E2 25410.827} C_VEL
LIN {X 0,Y 568.194,Z 603.452,A -85,B 0,C 180,E1 25407.568,E2 25407.568} C_VEL
LIN {X 0,Y 568.205,Z 603.459,A -85,B 0,C 180,E1 25404.205,E2 25404.205} C_VEL
LIN {X 0,Y 568.222,Z 603.451,A -85,B 0,C 180,E1 25400.874,E2 25400.874} C_VEL
LIN {X 0,Y 568.178,Z 603.457,A -85,B 0,C 180,E1 25397.618,E2 25397.618} C_VEL
LIN {X 0,Y 568.221,Z 603.457,A -85,B 0,C 180,E1 25394.365,E2 25394.365} C_VEL
LIN {X 0,Y 568.17,Z 603.457,A -85,B 0,C 180,E1 25391.161,E2 25391.161} C_VEL
LIN {X 0,Y 568.211,Z 603.461,A -85,B 0,C 180,E1 25387.889,E2 25387.889} C_VEL
LIN {X 0,Y 568.194,Z 603.714,A -85,B 0,C 180,E1 25385.061,E2 25385.061} C_VEL
LIN {X 0,Y 569.508,Z 610.42,A -85,B 0,C 180,E1 25384.275,E2 25384.275} C_VEL
LIN {X 0,Y 569.36,Z 638.458,A -85,B 0,C 180,E1 25381.107,E2 25381.107} C_VEL
LIN {X 0,Y 568.962,Z 667.012,A -85,B 0,C 180,E1 25377.784,E2 25377.784} C_VEL
LIN {X 0,Y 568.71,Z 692.669,A -85,B 0,C 180,E1 25374.893,E2 25374.893} C_VEL
LIN {X 0,Y 569.496,Z 699.413,A -85,B 0,C 180,E1 25374.767,E2 25374.767} C_VEL
LIN {X 0,Y 569.189,Z 826.523,A -85,B 0,C 180,E1 25373.137,E2 25373.137} C_VEL
LIN {X 0,Y 567.892,Z 835.229,A -85,B 0,C 180,E1 25373.02,E2 25373.02} C_VEL
LIN {X 0,Y 562.748,Z 850.955,A -85,B 0,C 180,E1 25372.742,E2 25372.742} C_VEL
LIN {X 0,Y 561.279,Z 858.286,A -85,B 0,C 180,E1 25372.516,E2 25372.516} C_VEL
LIN {X 0,Y 561.164,Z 860.318,A -85,B 0,C 180,E1 25372.436,E2 25372.436} C_VEL
LIN {X 0,Y 560.948,Z 874.975,A -85,B 0,C 180,E1 25371.75,E2 25371.75} C_VEL
LIN {X 0,Y 560.718,Z 889.315,A -85,B 0,C 180,E1 25370.868,E2 25370.868} C_VEL
LIN {X 0,Y 560.512,Z 902.692,A -85,B 0,C 180,E1 25369.828,E2 25369.828} C_VEL
LIN {X 0,Y 560.318,Z 914.496,A -85,B 0,C 180,E1 25368.68,E2 25368.68} C_VEL
LIN {X 0,Y 560.166,Z 924.987,A -85,B 0,C 180,E1 25367.422,E2 25367.422} C_VEL
LIN {X 0,Y 560.052,Z 934.139,A -85,B 0,C 180,E1 25366.053,E2 25366.053} C_VEL
LIN {X 0,Y 559.979,Z 941.966,A -85,B 0,C 180,E1 25364.571,E2 25364.571} C_VEL
LIN {X 0,Y 559.934,Z 948.289,A -85,B 0,C 180,E1 25362.971,E2 25362.971} C_VEL
LIN {X 0,Y 559.92,Z 952.781,A -85,B 0,C 180,E1 25361.358,E2 25361.358} C_VEL
LIN {X 0,Y 559.915,Z 955.469,A -85,B 0,C 180,E1 25359.73,E2 25359.73} C_VEL
LIN {X 0,Y 559.919,Z 956.499,A -85,B 0,C 180,E1 25357.975,E2 25357.975} C_VEL
LIN {X 0,Y 559.916,Z 955.608,A -85,B 0,C 180,E1 25356.31,E2 25356.31} C_VEL
LIN {X 0,Y 559.918,Z 952.935,A -85,B 0,C 180,E1 25354.623,E2 25354.623} C_VEL
LIN {X 0,Y 559.934,Z 948.512,A -85,B 0,C 180,E1 25353.006,E2 25353.006} C_VEL
LIN {X 0,Y 559.976,Z 942.286,A -85,B 0,C 180,E1 25351.411,E2 25351.411} C_VEL
LIN {X 0,Y 560.05,Z 934.33,A -85,B 0,C 180,E1 25349.889,E2 25349.889} C_VEL
LIN {X 0,Y 560.171,Z 924.833,A -85,B 0,C 180,E1 25348.467,E2 25348.467} C_VEL
LIN {X 0,Y 560.33,Z 913.734,A -85,B 0,C 180,E1 25347.148,E2 25347.148} C_VEL
LIN {X 0,Y 560.53,Z 901.722,A -85,B 0,C 180,E1 25345.998,E2 25345.998} C_VEL
LIN {X 0,Y 560.744,Z 887.688,A -85,B 0,C 180,E1 25344.93,E2 25344.93} C_VEL
LIN {X 0,Y 560.964,Z 873.783,A -85,B 0,C 180,E1 25344.097,E2 25344.097} C_VEL
LIN {X 0,Y 561.196,Z 858.161,A -85,B 0,C 180,E1 25343.387,E2 25343.387} C_VEL
LIN {X 0,Y 561.366,Z 842.519,A -85,B 0,C 180,E1 25342.882,E2 25342.882} C_VEL
LIN {X 0,Y 561.473,Z 825.522,A -85,B 0,C 180,E1 25342.543,E2 25342.543} C_VEL
LIN {X 0,Y 561.613,Z 697.249,A -85,B 0,C 180,E1 25340.871,E2 25340.871} C_VEL
LIN {X 0,Y 560.87,Z 692.389,A -85,B 0,C 180,E1 25340.755,E2 25340.755} C_VEL
LIN {X 0,Y 561.282,Z 666.515,A -85,B 0,C 180,E1 25337.741,E2 25337.741} C_VEL
LIN {X 0,Y 561.705,Z 636.526,A -85,B 0,C 180,E1 25334.249,E2 25334.249} C_VEL
LIN {X 0,Y 561.881,Z 611.6,A -85,B 0,C 180,E1 25331.383,E2 25331.383} C_VEL
LIN {X 0,Y 560.24,Z 604.566,A -85,B 0,C 180,E1 25330.461,E2 25330.461} C_VEL
LIN {X 0,Y 560.217,Z 604.437,A -85,B 0,C 180,E1 25327.08,E2 25327.08} C_VEL
LIN {X 0,Y 560.24,Z 604.45,A -85,B 0,C 180,E1 25324.084,E2 25324.084} C_VEL
LIN {X 0,Y 560.222,Z 604.445,A -85,B 0,C 180,E1 25320.812,E2 25320.812} C_VEL
LIN {X 0,Y 560.257,Z 604.448,A -85,B 0,C 180,E1 25317.725,E2 25317.725} C_VEL
LIN {X 0,Y 560.223,Z 604.437,A -85,B 0,C 180,E1 25314.461,E2 25314.461} C_VEL
LIN {X 0,Y 560.283,Z 604.443,A -85,B 0,C 180,E1 25311.24,E2 25311.24} C_VEL
LIN {X 0,Y 560.224,Z 604.447,A -85,B 0,C 180,E1 25307.959,E2 25307.959} C_VEL
LIN {X 0,Y 560.285,Z 604.445,A -85,B 0,C 180,E1 25304.679,E2 25304.679} C_VEL
LIN {X 0,Y 560.238,Z 604.453,A -85,B 0,C 180,E1 25301.426,E2 25301.426} C_VEL
LIN {X 0,Y 560.328,Z 604.764,A -85,B 0,C 180,E1 25300.773,E2 25300.773} C_VEL
LIN {X 0,Y 562.428,Z 613.842,A -85,B 0,C 180,E1 25299.517,E2 25299.517} C_VEL
LIN {X 0,Y 561.81,Z 640.07,A -85,B 0,C 180,E1 25296.335,E2 25296.335} C_VEL
LIN {X 0,Y 561.242,Z 668.24,A -85,B 0,C 180,E1 25292.962,E2 25292.962} C_VEL
LIN {X 0,Y 560.885,Z 692.604,A -85,B 0,C 180,E1 25290.145,E2 25290.145} C_VEL
LIN {X 0,Y 561.809,Z 700.315,A -85,B 0,C 180,E1 25289.992,E2 25289.992} C_VEL
LIN {X 0,Y 561.437,Z 832.679,A -85,B 0,C 180,E1 25288.249,E2 25288.249} C_VEL
LIN {X 0,Y 561.295,Z 849.665,A -85,B 0,C 180,E1 25287.821,E2 25287.821} C_VEL
LIN {X 0,Y 561.105,Z 864.907,A -85,B 0,C 180,E1 25287.243,E2 25287.243} C_VEL
LIN {X 0,Y 560.867,Z 880.711,A -85,B 0,C 180,E1 25286.423,E2 25286.423} C_VEL
LIN {X 0,Y 560.643,Z 894.416,A -85,B 0,C 180,E1 25285.5,E2 25285.5} C_VEL
LIN {X 0,Y 560.428,Z 907.7,A -85,B 0,C 180,E1 25284.369,E2 25284.369} C_VEL
LIN {X 0,Y 560.247,Z 919.337,A -85,B 0,C 180,E1 25283.133,E2 25283.133} C_VEL
LIN {X 0,Y 560.099,Z 930.155,A -85,B 0,C 180,E1 25281.686,E2 25281.686} C_VEL
LIN {X 0,Y 560.008,Z 938.703,A -85,B 0,C 180,E1 25280.235,E2 25280.235} C_VEL
LIN {X 0,Y 559.949,Z 945.981,A -85,B 0,C 180,E1 25278.613,E2 25278.613} C_VEL
LIN {X 0,Y 559.924,Z 951.22,A -85,B 0,C 180,E1 25276.997,E2 25276.997} C_VEL
LIN {X 0,Y 559.921,Z 954.7,A -85,B 0,C 180,E1 25275.311,E2 25275.311} C_VEL
LIN {X 0,Y 559.913,Z 956.361,A -85,B 0,C 180,E1 25273.612,E2 25273.612} C_VEL
LIN {X 0,Y 559.915,Z 956.114,A -85,B 0,C 180,E1 25271.898,E2 25271.898} C_VEL
LIN {X 0,Y 559.917,Z 954.131,A -85,B 0,C 180,E1 25270.234,E2 25270.234} C_VEL
LIN {X 0,Y 559.927,Z 950.449,A -85,B 0,C 180,E1 25268.637,E2 25268.637} C_VEL
LIN {X 0,Y 559.959,Z 944.735,A -85,B 0,C 180,E1 25266.981,E2 25266.981} C_VEL
LIN {X 0,Y 560.015,Z 937.954,A -85,B 0,C 180,E1 25265.53,E2 25265.53} C_VEL
LIN {X 0,Y 560.114,Z 929.082,A -85,B 0,C 180,E1 25264.065,E2 25264.065} C_VEL
LIN {X 0,Y 560.258,Z 918.701,A -85,B 0,C 180,E1 25262.7,E2 25262.7} C_VEL
LIN {X 0,Y 560.445,Z 906.59,A -85,B 0,C 180,E1 25261.437,E2 25261.437} C_VEL
LIN {X 0,Y 560.648,Z 894.238,A -85,B 0,C 180,E1 25260.396,E2 25260.396} C_VEL
LIN {X 0,Y 560.869,Z 880.328,A -85,B 0,C 180,E1 25259.465,E2 25259.465} C_VEL
LIN {X 0,Y 561.093,Z 865.548,A -85,B 0,C 180,E1 25258.697,E2 25258.697} C_VEL
LIN {X 0,Y 561.293,Z 850.099,A -85,B 0,C 180,E1 25258.102,E2 25258.102} C_VEL
LIN {X 0,Y 561.435,Z 833.288,A -85,B 0,C 180,E1 25257.673,E2 25257.673} C_VEL
LIN {X 0,Y 561.584,Z 781.644,A -85,B 0,C 180,E1 25256.973,E2 25256.973} C_VEL
LIN {X 0,Y 561.603,Z 697.151,A -85,B 0,C 180,E1 25255.87,E2 25255.87} C_VEL
LIN {X 0,Y 560.885,Z 692.331,A -85,B 0,C 180,E1 25255.746,E2 25255.746} C_VEL
LIN {X 0,Y 561.308,Z 666.581,A -85,B 0,C 180,E1 25252.725,E2 25252.725} C_VEL
LIN {X 0,Y 561.928,Z 637.832,A -85,B 0,C 180,E1 25249.288,E2 25249.288} C_VEL
LIN {X 0,Y 562.495,Z 613.001,A -85,B 0,C 180,E1 25246.254,E2 25246.254} C_VEL
LIN {X 0,Y 560.292,Z 604.563,A -85,B 0,C 180,E1 25245.035,E2 25245.035} C_VEL
LIN {X 0,Y 560.269,Z 604.444,A -85,B 0,C 180,E1 25241.596,E2 25241.596} C_VEL
LIN {X 0,Y 560.267,Z 604.446,A -85,B 0,C 180,E1 25238.393,E2 25238.393} C_VEL
LIN {X 0,Y 560.264,Z 604.444,A -85,B 0,C 180,E1 25235.075,E2 25235.075} C_VEL
LIN {X 0,Y 560.266,Z 604.44,A -85,B 0,C 180,E1 25231.767,E2 25231.767} C_VEL
LIN {X 0,Y 560.28,Z 604.445,A -85,B 0,C 180,E1 25228.383,E2 25228.383} C_VEL
LIN {X 0,Y 560.274,Z 604.438,A -85,B 0,C 180,E1 25224.965,E2 25224.965} C_VEL
LIN {X 0,Y 560.263,Z 604.444,A -85,B 0,C 180,E1 25221.598,E2 25221.598} C_VEL
LIN {X 0,Y 560.266,Z 604.441,A -85,B 0,C 180,E1 25218.303,E2 25218.303} C_VEL
LIN {X 0,Y 560.262,Z 604.438,A -85,B 0,C 180,E1 25214.997,E2 25214.997} C_VEL
LIN {X 0,Y 560.277,Z 604.448,A -85,B 0,C 180,E1 25211.634,E2 25211.634} C_VEL
LIN {X 0,Y 560.276,Z 604.439,A -85,B 0,C 180,E1 25208.208,E2 25208.208} C_VEL
LIN {X 0,Y 560.26,Z 604.443,A -85,B 0,C 180,E1 25204.914,E2 25204.914} C_VEL
LIN {X 0,Y 560.269,Z 604.442,A -85,B 0,C 180,E1 25201.636,E2 25201.636} C_VEL
LIN {X 0,Y 560.257,Z 604.442,A -85,B 0,C 180,E1 25198.364,E2 25198.364} C_VEL
LIN {X 0,Y 560.278,Z 604.442,A -85,B 0,C 180,E1 25194.984,E2 25194.984} C_VEL
LIN {X 0,Y 560.281,Z 604.436,A -85,B 0,C 180,E1 25191.586,E2 25191.586} C_VEL
LIN {X 0,Y 560.258,Z 604.444,A -85,B 0,C 180,E1 25188.261,E2 25188.261} C_VEL
LIN {X 0,Y 560.271,Z 604.439,A -85,B 0,C 180,E1 25185.003,E2 25185.003} C_VEL
LIN {X 0,Y 560.252,Z 604.438,A -85,B 0,C 180,E1 25181.702,E2 25181.702} C_VEL
LIN {X 0,Y 560.281,Z 604.448,A -85,B 0,C 180,E1 25178.321,E2 25178.321} C_VEL
LIN {X 0,Y 560.279,Z 604.439,A -85,B 0,C 180,E1 25174.867,E2 25174.867} C_VEL
LIN {X 0,Y 560.254,Z 604.445,A -85,B 0,C 180,E1 25171.543,E2 25171.543} C_VEL
LIN {X 0,Y 560.276,Z 604.439,A -85,B 0,C 180,E1 25168.234,E2 25168.234} C_VEL
LIN {X 0,Y 560.251,Z 604.441,A -85,B 0,C 180,E1 25164.924,E2 25164.924} C_VEL
LIN {X 0,Y 560.283,Z 604.445,A -85,B 0,C 180,E1 25161.575,E2 25161.575} C_VEL
LIN {X 0,Y 560.273,Z 604.439,A -85,B 0,C 180,E1 25158.241,E2 25158.241} C_VEL
LIN {X 0,Y 560.251,Z 604.446,A -85,B 0,C 180,E1 25154.886,E2 25154.886} C_VEL
LIN {X 0,Y 560.278,Z 604.443,A -85,B 0,C 180,E1 25151.595,E2 25151.595} C_VEL
LIN {X 0,Y 560.245,Z 604.445,A -85,B 0,C 180,E1 25148.394,E2 25148.394} C_VEL
LIN {X 0,Y 560.279,Z 604.442,A -85,B 0,C 180,E1 25145.074,E2 25145.074} C_VEL
LIN {X 0,Y 560.32,Z 604.724,A -85,B 0,C 180,E1 25143.34,E2 25143.34} C_VEL
LIN {X 0,Y 564.667,Z 617.36,A -85,B 0,C 180,E1 25142.027,E2 25142.027} C_VEL
LIN {X 0,Y 563.769,Z 661.008,A -85,B 0,C 180,E1 25138.726,E2 25138.726} C_VEL
LIN {X 0,Y 562.927,Z 704.317,A -85,B 0,C 180,E1 25135.538,E2 25135.538} C_VEL
LIN {X 0,Y 562.875,Z 709.31,A -85,B 0,C 180,E1 25135.188,E2 25135.188} C_VEL
LIN {X 0,Y 564.005,Z 717.916,A -85,B 0,C 180,E1 25135.001,E2 25135.001} C_VEL
LIN {X 0,Y 563.114,Z 927.53,A -85,B 0,C 180,E1 25132.157,E2 25132.157} C_VEL
LIN {X 0,Y 562.878,Z 946.926,A -85,B 0,C 180,E1 25131.698,E2 25131.698} C_VEL
LIN {X 0,Y 562.583,Z 965.066,A -85,B 0,C 180,E1 25131.083,E2 25131.083} C_VEL
LIN {X 0,Y 562.216,Z 983.451,A -85,B 0,C 180,E1 25130.256,E2 25130.256} C_VEL
LIN {X 0,Y 561.827,Z 1000.716,A -85,B 0,C 180,E1 25129.276,E2 25129.276} C_VEL
LIN {X 0,Y 561.427,Z 1017.467,A -85,B 0,C 180,E1 25128.105,E2 25128.105} C_VEL
LIN {X 0,Y 561.049,Z 1033.105,A -85,B 0,C 180,E1 25126.78,E2 25126.78} C_VEL
LIN {X 0,Y 560.735,Z 1046.685,A -85,B 0,C 180,E1 25125.407,E2 25125.407} C_VEL
LIN {X 0,Y 560.458,Z 1059.752,A -85,B 0,C 180,E1 25123.831,E2 25123.831} C_VEL
LIN {X 0,Y 560.246,Z 1071.296,A -85,B 0,C 180,E1 25122.157,E2 25122.157} C_VEL
LIN {X 0,Y 560.097,Z 1081.344,A -85,B 0,C 180,E1 25120.385,E2 25120.385} C_VEL
LIN {X 0,Y 560.007,Z 1089.433,A -85,B 0,C 180,E1 25118.625,E2 25118.625} C_VEL
LIN {X 0,Y 559.942,Z 1096.129,A -85,B 0,C 180,E1 25116.768,E2 25116.768} C_VEL
LIN {X 0,Y 559.923,Z 1101.297,A -85,B 0,C 180,E1 25114.814,E2 25114.814} C_VEL
LIN {X 0,Y 559.906,Z 1104.661,A -85,B 0,C 180,E1 25112.866,E2 25112.866} C_VEL
LIN {X 0,Y 559.91,Z 1106.305,A -85,B 0,C 180,E1 25110.921,E2 25110.921} C_VEL
LIN {X 0,Y 559.907,Z 1106.263,A -85,B 0,C 180,E1 25108.977,E2 25108.977} C_VEL
LIN {X 0,Y 559.909,Z 1104.538,A -85,B 0,C 180,E1 25107.031,E2 25107.031} C_VEL
LIN {X 0,Y 559.921,Z 1101.086,A -85,B 0,C 180,E1 25105.083,E2 25105.083} C_VEL
LIN {X 0,Y 559.945,Z 1095.814,A -85,B 0,C 180,E1 25103.127,E2 25103.127} C_VEL
LIN {X 0,Y 560.011,Z 1088.593,A -85,B 0,C 180,E1 25101.167,E2 25101.167} C_VEL
LIN {X 0,Y 560.121,Z 1079.735,A -85,B 0,C 180,E1 25099.301,E2 25099.301} C_VEL
LIN {X 0,Y 560.277,Z 1069.311,A -85,B 0,C 180,E1 25097.529,E2 25097.529} C_VEL
LIN {X 0,Y 560.505,Z 1057.324,A -85,B 0,C 180,E1 25095.854,E2 25095.854} C_VEL
LIN {X 0,Y 560.79,Z 1044.159,A -85,B 0,C 180,E1 25094.321,E2 25094.321} C_VEL
LIN {X 0,Y 561.131,Z 1029.584,A -85,B 0,C 180,E1 25092.902,E2 25092.902} C_VEL
LIN {X 0,Y 561.507,Z 1013.893,A -85,B 0,C 180,E1 25091.628,E2 25091.628} C_VEL
LIN {X 0,Y 561.89,Z 997.182,A -85,B 0,C 180,E1 25090.509,E2 25090.509} C_VEL
LIN {X 0,Y 562.279,Z 979.428,A -85,B 0,C 180,E1 25089.548,E2 25089.548} C_VEL
LIN {X 0,Y 562.625,Z 961.275,A -85,B 0,C 180,E1 25088.777,E2 25088.777} C_VEL
LIN {X 0,Y 562.924,Z 942.161,A -85,B 0,C 180,E1 25088.174,E2 25088.174} C_VEL
LIN {X 0,Y 563.148,Z 922.549,A -85,B 0,C 180,E1 25087.762,E2 25087.762} C_VEL
LIN {X 0,Y 563.853,Z 715.407,A -85,B 0,C 180,E1 25084.957,E2 25084.957} C_VEL
LIN {X 0,Y 562.874,Z 709.296,A -85,B 0,C 180,E1 25084.812,E2 25084.812} C_VEL
LIN {X 0,Y 563.638,Z 667.891,A -85,B 0,C 180,E1 25081.786,E2 25081.786} C_VEL
LIN {X 0,Y 564.543,Z 623.176,A -85,B 0,C 180,E1 25078.418,E2 25078.418} C_VEL
LIN {X 0,Y 564.546,Z 616.585,A -85,B 0,C 180,E1 25077.905,E2 25077.905} C_VEL
LIN {X 0,Y 560.32,Z 604.73,A -85,B 0,C 180,E1 25076.659,E2 25076.659} C_VEL
LIN {X 0,Y 560.275,Z 604.439,A -85,B 0,C 180,E1 25074.8,E2 25074.8} C_VEL
LIN {X 0,Y 560.258,Z 604.448,A -85,B 0,C 180,E1 25071.476,E2 25071.476} C_VEL
LIN {X 0,Y 560.276,Z 604.439,A -85,B 0,C 180,E1 25068.088,E2 25068.088} C_VEL
LIN {X 0,Y 560.271,Z 604.445,A -85,B 0,C 180,E1 25064.679,E2 25064.679} C_VEL
LIN {X 0,Y 560.265,Z 604.442,A -85,B 0,C 180,E1 25061.449,E2 25061.449} C_VEL
LIN {X 0,Y 560.261,Z 604.444,A -85,B 0,C 180,E1 25058.257,E2 25058.257} C_VEL
LIN {X 0,Y 560.272,Z 604.445,A -85,B 0,C 180,E1 25054.949,E2 25054.949} C_VEL
LIN {X 0,Y 560.266,Z 604.44,A -85,B 0,C 180,E1 25051.646,E2 25051.646} C_VEL
LIN {X 0,Y 560.262,Z 604.447,A -85,B 0,C 180,E1 25048.224,E2 25048.224} C_VEL
LIN {X 0,Y 560.279,Z 604.442,A -85,B 0,C 180,E1 25044.908,E2 25044.908} C_VEL
LIN {X 0,Y 560.243,Z 604.445,A -85,B 0,C 180,E1 25041.68,E2 25041.68} C_VEL
LIN {X 0,Y 560.281,Z 604.446,A -85,B 0,C 180,E1 25038.413,E2 25038.413} C_VEL
LIN {X 0,Y 560.237,Z 604.445,A -85,B 0,C 180,E1 25035.21,E2 25035.21} C_VEL
LIN {X 0,Y 560.257,Z 604.45,A -85,B 0,C 180,E1 25031.843,E2 25031.843} C_VEL
LIN {X 0,Y 560.245,Z 604.446,A -85,B 0,C 180,E1 25028.725,E2 25028.725} C_VEL
LIN {X 0,Y 560.232,Z 604.484,A -85,B 0,C 180,E1 25025.351,E2 25025.351} C_VEL
LIN {X 0,Y 560.733,Z 606.846,A -85,B 0,C 180,E1 25025.012,E2 25025.012} C_VEL
LIN {X 0,Y 561.777,Z 612.174,A -85,B 0,C 180,E1 25024.389,E2 25024.389} C_VEL
LIN {X 0,Y 561.687,Z 640.47,A -85,B 0,C 180,E1 25021.224,E2 25021.224} C_VEL
LIN {X 0,Y 561.345,Z 665.015,A -85,B 0,C 180,E1 25018.367,E2 25018.367} C_VEL
LIN {X 0,Y 560.868,Z 691.66,A -85,B 0,C 180,E1 25015.229,E2 25015.229} C_VEL
LIN {X 0,Y 561.015,Z 693.654,A -85,B 0,C 180,E1 25015.105,E2 25015.105} C_VEL
LIN {X 0,Y 561.835,Z 700.494,A -85,B 0,C 180,E1 25014.989,E2 25014.989} C_VEL
LIN {X 0,Y 561.438,Z 832.852,A -85,B 0,C 180,E1 25013.247,E2 25013.247} C_VEL
LIN {X 0,Y 561.293,Z 849.91,A -85,B 0,C 180,E1 25012.814,E2 25012.814} C_VEL
LIN {X 0,Y 561.164,Z 860.318,A -85,B 0,C 180,E1 25012.436,E2 25012.436} C_VEL
LIN {X 0,Y 560.095,Z 867.532,A -85,B 0,C 180,E1 25012.149,E2 25012.149} C_VEL
LIN {X 0,Y 555.186,Z 881.184,A -85,B 0,C 180,E1 25011.536,E2 25011.536} C_VEL
LIN {X 0,Y 553.089,Z 888.663,A -85,B 0,C 180,E1 25011.096,E2 25011.096} C_VEL
LIN {X 0,Y 552.838,Z 891.396,A -85,B 0,C 180,E1 25010.908,E2 25010.908} C_VEL
LIN {X 0,Y 552.589,Z 904.423,A -85,B 0,C 180,E1 25009.842,E2 25009.842} C_VEL
LIN {X 0,Y 552.367,Z 916.445,A -85,B 0,C 180,E1 25008.62,E2 25008.62} C_VEL
LIN {X 0,Y 552.178,Z 927.285,A -85,B 0,C 180,E1 25007.237,E2 25007.237} C_VEL
LIN {X 0,Y 552.058,Z 936.01,A -85,B 0,C 180,E1 25005.847,E2 25005.847} C_VEL
LIN {X 0,Y 551.978,Z 943.38,A -85,B 0,C 180,E1 25004.341,E2 25004.341} C_VEL
LIN {X 0,Y 551.935,Z 949.444,A -85,B 0,C 180,E1 25002.687,E2 25002.687} C_VEL
LIN {X 0,Y 551.918,Z 953.649,A -85,B 0,C 180,E1 25000.968,E2 25000.968} C_VEL
LIN {X 0,Y 551.914,Z 955.93,A -85,B 0,C 180,E1 24999.313,E2 24999.313} C_VEL
LIN {X 0,Y 551.914,Z 956.439,A -85,B 0,C 180,E1 24997.639,E2 24997.639} C_VEL
LIN {X 0,Y 551.916,Z 955.23,A -85,B 0,C 180,E1 24995.932,E2 24995.932} C_VEL
LIN {X 0,Y 551.921,Z 952.133,A -85,B 0,C 180,E1 24994.228,E2 24994.228} C_VEL
LIN {X 0,Y 551.948,Z 947.332,A -85,B 0,C 180,E1 24992.579,E2 24992.579} C_VEL
LIN {X 0,Y 552.003,Z 940.617,A -85,B 0,C 180,E1 24990.959,E2 24990.959} C_VEL
LIN {X 0,Y 552.101,Z 932.906,A -85,B 0,C 180,E1 24989.53,E2 24989.53} C_VEL
LIN {X 0,Y 552.25,Z 922.958,A -85,B 0,C 180,E1 24988.084,E2 24988.084} C_VEL
LIN {X 0,Y 552.449,Z 912.027,A -85,B 0,C 180,E1 24986.808,E2 24986.808} C_VEL
LIN {X 0,Y 552.686,Z 899.481,A -85,B 0,C 180,E1 24985.636,E2 24985.636} C_VEL
LIN {X 0,Y 552.94,Z 886.201,A -85,B 0,C 180,E1 24984.64,E2 24984.64} C_VEL
LIN {X 0,Y 553.208,Z 871.313,A -85,B 0,C 180,E1 24983.771,E2 24983.771} C_VEL
LIN {X 0,Y 553.462,Z 856.437,A -85,B 0,C 180,E1 24983.111,E2 24983.111} C_VEL
LIN {X 0,Y 553.657,Z 839.746,A -85,B 0,C 180,E1 24982.596,E2 24982.596} C_VEL
LIN {X 0,Y 553.771,Z 823.147,A -85,B 0,C 180,E1 24982.29,E2 24982.29} C_VEL
LIN {X 0,Y 553.964,Z 698.218,A -85,B 0,C 180,E1 24980.641,E2 24980.641} C_VEL
LIN {X 0,Y 553.126,Z 692.857,A -85,B 0,C 180,E1 24980.511,E2 24980.511} C_VEL
LIN {X 0,Y 553.636,Z 665.049,A -85,B 0,C 180,E1 24977.23,E2 24977.23} C_VEL
LIN {X 0,Y 554.064,Z 636.285,A -85,B 0,C 180,E1 24973.866,E2 24973.866} C_VEL
LIN {X 0,Y 554.195,Z 613.631,A -85,B 0,C 180,E1 24971.256,E2 24971.256} C_VEL
LIN {X 0,Y 552.328,Z 605.572,A -85,B 0,C 180,E1 24970.207,E2 24970.207} C_VEL
LIN {X 0,Y 552.272,Z 605.425,A -85,B 0,C 180,E1 24966.947,E2 24966.947} C_VEL
LIN {X 0,Y 552.333,Z 605.433,A -85,B 0,C 180,E1 24963.762,E2 24963.762} C_VEL
LIN {X 0,Y 552.276,Z 605.435,A -85,B 0,C 180,E1 24960.58,E2 24960.58} C_VEL
LIN {X 0,Y 552.345,Z 605.434,A -85,B 0,C 180,E1 24957.374,E2 24957.374} C_VEL
LIN {X 0,Y 552.28,Z 605.426,A -85,B 0,C 180,E1 24954.152,E2 24954.152} C_VEL
LIN {X 0,Y 552.337,Z 605.427,A -85,B 0,C 180,E1 24950.893,E2 24950.893} C_VEL
LIN {X 0,Y 552.292,Z 605.438,A -85,B 0,C 180,E1 24947.707,E2 24947.707} C_VEL
LIN {X 0,Y 552.305,Z 605.436,A -85,B 0,C 180,E1 24944.253,E2 24944.253} C_VEL
LIN {X 0,Y 552.352,Z 605.666,A -85,B 0,C 180,E1 24941.145,E2 24941.145} C_VEL
LIN {X 0,Y 554.875,Z 616.251,A -85,B 0,C 180,E1 24939.648,E2 24939.648} C_VEL
LIN {X 0,Y 554.16,Z 643.429,A -85,B 0,C 180,E1 24936.319,E2 24936.319} C_VEL
LIN {X 0,Y 553.549,Z 670.877,A -85,B 0,C 180,E1 24933.003,E2 24933.003} C_VEL
LIN {X 0,Y 553.173,Z 692.834,A -85,B 0,C 180,E1 24930.427,E2 24930.427} C_VEL
LIN {X 0,Y 554.244,Z 701.077,A -85,B 0,C 180,E1 24930.252,E2 24930.252} C_VEL
LIN {X 0,Y 553.715,Z 833.044,A -85,B 0,C 180,E1 24928.461,E2 24928.461} C_VEL
LIN {X 0,Y 553.547,Z 850.004,A -85,B 0,C 180,E1 24928.024,E2 24928.024} C_VEL
LIN {X 0,Y 553.335,Z 864.579,A -85,B 0,C 180,E1 24927.463,E2 24927.463} C_VEL
LIN {X 0,Y 553.071,Z 879.569,A -85,B 0,C 180,E1 24926.684,E2 24926.684} C_VEL
LIN {X 0,Y 552.797,Z 893.567,A -85,B 0,C 180,E1 24925.747,E2 24925.747} C_VEL
LIN {X 0,Y 552.541,Z 906.997,A -85,B 0,C 180,E1 24924.601,E2 24924.601} C_VEL
LIN {X 0,Y 552.324,Z 918.798,A -85,B 0,C 180,E1 24923.347,E2 24923.347} C_VEL
LIN {X 0,Y 552.154,Z 929.004,A -85,B 0,C 180,E1 24921.985,E2 24921.985} C_VEL
LIN {X 0,Y 552.036,Z 937.814,A -85,B 0,C 180,E1 24920.513,E2 24920.513} C_VEL
LIN {X 0,Y 551.966,Z 944.656,A -85,B 0,C 180,E1 24919.036,E2 24919.036} C_VEL
LIN {X 0,Y 551.931,Z 950.443,A -85,B 0,C 180,E1 24917.338,E2 24917.338} C_VEL
LIN {X 0,Y 551.917,Z 954.096,A -85,B 0,C 180,E1 24915.737,E2 24915.737} C_VEL
LIN {X 0,Y 551.914,Z 956.121,A -85,B 0,C 180,E1 24914.016,E2 24914.016} C_VEL
LIN {X 0,Y 551.914,Z 956.358,A -85,B 0,C 180,E1 24912.281,E2 24912.281} C_VEL
LIN {X 0,Y 551.915,Z 954.815,A -85,B 0,C 180,E1 24910.639,E2 24910.639} C_VEL
LIN {X 0,Y 551.93,Z 951.257,A -85,B 0,C 180,E1 24908.869,E2 24908.869} C_VEL
LIN {X 0,Y 551.955,Z 946.325,A -85,B 0,C 180,E1 24907.304,E2 24907.304} C_VEL
LIN {X 0,Y 552.021,Z 939.123,A -85,B 0,C 180,E1 24905.654,E2 24905.654} C_VEL
LIN {X 0,Y 552.132,Z 930.587,A -85,B 0,C 180,E1 24904.162,E2 24904.162} C_VEL
LIN {X 0,Y 552.298,Z 920.186,A -85,B 0,C 180,E1 24902.734,E2 24902.734} C_VEL
LIN {X 0,Y 552.501,Z 909.208,A -85,B 0,C 180,E1 24901.52,E2 24901.52} C_VEL
LIN {X 0,Y 552.742,Z 896.671,A -85,B 0,C 180,E1 24900.408,E2 24900.408} C_VEL
LIN {X 0,Y 553.017,Z 882.571,A -85,B 0,C 180,E1 24899.406,E2 24899.406} C_VEL
LIN {X 0,Y 553.267,Z 867.954,A -85,B 0,C 180,E1 24898.605,E2 24898.605} C_VEL
LIN {X 0,Y 553.515,Z 852.391,A -85,B 0,C 180,E1 24897.967,E2 24897.967} C_VEL
LIN {X 0,Y 553.697,Z 836.373,A -85,B 0,C 180,E1 24897.517,E2 24897.517} C_VEL
LIN {X 0,Y 553.824,Z 812.72,A -85,B 0,C 180,E1 24897.151,E2 24897.151} C_VEL
LIN {X 0,Y 554.059,Z 698.092,A -85,B 0,C 180,E1 24895.603,E2 24895.603} C_VEL
LIN {X 0,Y 553.16,Z 692.461,A -85,B 0,C 180,E1 24895.448,E2 24895.448} C_VEL
LIN {X 0,Y 553.743,Z 664.467,A -85,B 0,C 180,E1 24892.099,E2 24892.099} C_VEL
LIN {X 0,Y 554.42,Z 636.959,A -85,B 0,C 180,E1 24888.767,E2 24888.767} C_VEL
LIN {X 0,Y 554.887,Z 615.152,A -85,B 0,C 180,E1 24886.074,E2 24886.074} C_VEL
LIN {X 0,Y 552.343,Z 605.534,A -85,B 0,C 180,E1 24884.65,E2 24884.65} C_VEL
LIN {X 0,Y 552.324,Z 605.435,A -85,B 0,C 180,E1 24881.3,E2 24881.3} C_VEL
LIN {X 0,Y 552.329,Z 605.431,A -85,B 0,C 180,E1 24877.988,E2 24877.988} C_VEL
LIN {X 0,Y 552.337,Z 605.436,A -85,B 0,C 180,E1 24874.548,E2 24874.548} C_VEL
LIN {X 0,Y 552.331,Z 605.428,A -85,B 0,C 180,E1 24871.102,E2 24871.102} C_VEL
LIN {X 0,Y 552.325,Z 605.434,A -85,B 0,C 180,E1 24867.843,E2 24867.843} C_VEL
LIN {X 0,Y 552.329,Z 605.431,A -85,B 0,C 180,E1 24864.491,E2 24864.491} C_VEL
LIN {X 0,Y 552.333,Z 605.428,A -85,B 0,C 180,E1 24861.115,E2 24861.115} C_VEL
LIN {X 0,Y 552.335,Z 605.436,A -85,B 0,C 180,E1 24857.706,E2 24857.706} C_VEL
LIN {X 0,Y 552.332,Z 605.426,A -85,B 0,C 180,E1 24854.36,E2 24854.36} C_VEL
LIN {X 0,Y 552.321,Z 605.429,A -85,B 0,C 180,E1 24851.063,E2 24851.063} C_VEL
LIN {X 0,Y 552.334,Z 605.434,A -85,B 0,C 180,E1 24847.699,E2 24847.699} C_VEL
LIN {X 0,Y 552.332,Z 605.427,A -85,B 0,C 180,E1 24844.361,E2 24844.361} C_VEL
LIN {X 0,Y 552.327,Z 605.431,A -85,B 0,C 180,E1 24840.934,E2 24840.934} C_VEL
LIN {X 0,Y 552.334,Z 605.43,A -85,B 0,C 180,E1 24837.614,E2 24837.614} C_VEL
LIN {X 0,Y 552.318,Z 605.431,A -85,B 0,C 180,E1 24834.286,E2 24834.286} C_VEL
LIN {X 0,Y 552.337,Z 605.431,A -85,B 0,C 180,E1 24830.939,E2 24830.939} C_VEL
LIN {X 0,Y 552.336,Z 605.427,A -85,B 0,C 180,E1 24827.56,E2 24827.56} C_VEL
LIN {X 0,Y 552.319,Z 605.435,A -85,B 0,C 180,E1 24824.136,E2 24824.136} C_VEL
LIN {X 0,Y 552.335,Z 605.425,A -85,B 0,C 180,E1 24820.874,E2 24820.874} C_VEL
LIN {X 0,Y 552.313,Z 605.429,A -85,B 0,C 180,E1 24817.656,E2 24817.656} C_VEL
LIN {X 0,Y 552.337,Z 605.434,A -85,B 0,C 180,E1 24814.355,E2 24814.355} C_VEL
LIN {X 0,Y 552.325,Z 605.43,A -85,B 0,C 180,E1 24810.978,E2 24810.978} C_VEL
LIN {X 0,Y 552.32,Z 605.436,A -85,B 0,C 180,E1 24807.476,E2 24807.476} C_VEL
LIN {X 0,Y 552.339,Z 605.429,A -85,B 0,C 180,E1 24804.192,E2 24804.192} C_VEL
LIN {X 0,Y 552.31,Z 605.434,A -85,B 0,C 180,E1 24800.951,E2 24800.951} C_VEL
LIN {X 0,Y 552.34,Z 605.435,A -85,B 0,C 180,E1 24797.61,E2 24797.61} C_VEL
LIN {X 0,Y 552.316,Z 605.431,A -85,B 0,C 180,E1 24794.329,E2 24794.329} C_VEL
LIN {X 0,Y 552.328,Z 605.437,A -85,B 0,C 180,E1 24790.943,E2 24790.943} C_VEL
LIN {X 0,Y 552.343,Z 605.431,A -85,B 0,C 180,E1 24787.545,E2 24787.545} C_VEL
LIN {X 0,Y 552.306,Z 605.432,A -85,B 0,C 180,E1 24784.175,E2 24784.175} C_VEL
LIN {X 0,Y 552.383,Z 605.833,A -85,B 0,C 180,E1 24783.743,E2 24783.743} C_VEL
LIN {X 0,Y 557.482,Z 620.422,A -85,B 0,C 180,E1 24782.247,E2 24782.247} C_VEL
LIN {X 0,Y 556.427,Z 664.071,A -85,B 0,C 180,E1 24778.906,E2 24778.906} C_VEL
LIN {X 0,Y 555.448,Z 706.954,A -85,B 0,C 180,E1 24775.71,E2 24775.71} C_VEL
LIN {X 0,Y 555.541,Z 710.167,A -85,B 0,C 180,E1 24775.521,E2 24775.521} C_VEL
LIN {X 0,Y 556.751,Z 719.098,A -85,B 0,C 180,E1 24775.333,E2 24775.333} C_VEL
LIN {X 0,Y 555.704,Z 927.53,A -85,B 0,C 180,E1 24772.468,E2 24772.468} C_VEL
LIN {X 0,Y 555.425,Z 946.933,A -85,B 0,C 180,E1 24772.004,E2 24772.004} C_VEL
LIN {X 0,Y 555.066,Z 965.502,A -85,B 0,C 180,E1 24771.363,E2 24771.363} C_VEL
LIN {X 0,Y 554.634,Z 983.813,A -85,B 0,C 180,E1 24770.526,E2 24770.526} C_VEL
LIN {X 0,Y 554.185,Z 1000.713,A -85,B 0,C 180,E1 24769.553,E2 24769.553} C_VEL
LIN {X 0,Y 553.716,Z 1017.465,A -85,B 0,C 180,E1 24768.367,E2 24768.367} C_VEL
LIN {X 0,Y 553.269,Z 1033.104,A -85,B 0,C 180,E1 24767.023,E2 24767.023} C_VEL
LIN {X 0,Y 552.894,Z 1046.685,A -85,B 0,C 180,E1 24765.631,E2 24765.631} C_VEL
LIN {X 0,Y 552.567,Z 1059.753,A -85,B 0,C 180,E1 24764.032,E2 24764.032} C_VEL
LIN {X 0,Y 552.314,Z 1071.297,A -85,B 0,C 180,E1 24762.334,E2 24762.334} C_VEL
LIN {X 0,Y 552.134,Z 1081.334,A -85,B 0,C 180,E1 24760.539,E2 24760.539} C_VEL
LIN {X 0,Y 552.023,Z 1089.433,A -85,B 0,C 180,E1 24758.751,E2 24758.751} C_VEL
LIN {X 0,Y 551.949,Z 1096.129,A -85,B 0,C 180,E1 24756.866,E2 24756.866} C_VEL
LIN {X 0,Y 551.923,Z 1101.297,A -85,B 0,C 180,E1 24754.884,E2 24754.884} C_VEL
LIN {X 0,Y 551.907,Z 1104.66,A -85,B 0,C 180,E1 24752.907,E2 24752.907} C_VEL
LIN {X 0,Y 551.91,Z 1106.305,A -85,B 0,C 180,E1 24750.934,E2 24750.934} C_VEL
LIN {X 0,Y 551.907,Z 1106.264,A -85,B 0,C 180,E1 24748.962,E2 24748.962} C_VEL
LIN {X 0,Y 551.91,Z 1104.538,A -85,B 0,C 180,E1 24746.988,E2 24746.988} C_VEL
LIN {X 0,Y 551.922,Z 1101.086,A -85,B 0,C 180,E1 24745.011,E2 24745.011} C_VEL
LIN {X 0,Y 551.953,Z 1095.818,A -85,B 0,C 180,E1 24743.029,E2 24743.029} C_VEL
LIN {X 0,Y 552.027,Z 1088.593,A -85,B 0,C 180,E1 24741.038,E2 24741.038} C_VEL
LIN {X 0,Y 552.161,Z 1079.734,A -85,B 0,C 180,E1 24739.145,E2 24739.145} C_VEL
LIN {X 0,Y 552.353,Z 1069.259,A -85,B 0,C 180,E1 24737.34,E2 24737.34} C_VEL
LIN {X 0,Y 552.626,Z 1057.323,A -85,B 0,C 180,E1 24735.648,E2 24735.648} C_VEL
LIN {X 0,Y 552.955,Z 1044.671,A -85,B 0,C 180,E1 24734.147,E2 24734.147} C_VEL
LIN {X 0,Y 553.353,Z 1030.266,A -85,B 0,C 180,E1 24732.715,E2 24732.715} C_VEL
LIN {X 0,Y 553.796,Z 1014.625,A -85,B 0,C 180,E1 24731.418,E2 24731.418} C_VEL
LIN {X 0,Y 554.246,Z 998.076,A -85,B 0,C 180,E1 24730.284,E2 24730.284} C_VEL
LIN {X 0,Y 554.701,Z 980.536,A -85,B 0,C 180,E1 24729.31,E2 24729.31} C_VEL
LIN {X 0,Y 555.112,Z 962.504,A -85,B 0,C 180,E1 24728.522,E2 24728.522} C_VEL
LIN {X 0,Y 555.465,Z 943.735,A -85,B 0,C 180,E1 24727.908,E2 24727.908} C_VEL
LIN {X 0,Y 555.728,Z 924.797,A -85,B 0,C 180,E1 24727.485,E2 24727.485} C_VEL
LIN {X 0,Y 556.6,Z 716.545,A -85,B 0,C 180,E1 24724.624,E2 24724.624} C_VEL
LIN {X 0,Y 555.438,Z 709.363,A -85,B 0,C 180,E1 24724.455,E2 24724.455} C_VEL
LIN {X 0,Y 556.339,Z 667.891,A -85,B 0,C 180,E1 24721.382,E2 24721.382} C_VEL
LIN {X 0,Y 557.386,Z 624.213,A -85,B 0,C 180,E1 24718.047,E2 24718.047} C_VEL
LIN {X 0,Y 557.319,Z 619.53,A -85,B 0,C 180,E1 24717.672,E2 24717.672} C_VEL
LIN {X 0,Y 552.368,Z 605.747,A -85,B 0,C 180,E1 24716.24,E2 24716.24} C_VEL
LIN {X 0,Y 552.334,Z 605.424,A -85,B 0,C 180,E1 24715.234,E2 24715.234} C_VEL
LIN {X 0,Y 552.317,Z 605.435,A -85,B 0,C 180,E1 24711.879,E2 24711.879} C_VEL
LIN {X 0,Y 552.333,Z 605.433,A -85,B 0,C 180,E1 24708.643,E2 24708.643} C_VEL
LIN {X 0,Y 552.323,Z 605.432,A -85,B 0,C 180,E1 24705.352,E2 24705.352} C_VEL
LIN {X 0,Y 552.335,Z 605.429,A -85,B 0,C 180,E1 24702.051,E2 24702.051} C_VEL
LIN {X 0,Y 552.338,Z 605.435,A -85,B 0,C 180,E1 24698.648,E2 24698.648} C_VEL
LIN {X 0,Y 552.332,Z 605.431,A -85,B 0,C 180,E1 24695.271,E2 24695.271} C_VEL
LIN {X 0,Y 552.317,Z 605.433,A -85,B 0,C 180,E1 24692.034,E2 24692.034} C_VEL
LIN {X 0,Y 552.34,Z 605.435,A -85,B 0,C 180,E1 24688.666,E2 24688.666} C_VEL
LIN {X 0,Y 552.331,Z 605.429,A -85,B 0,C 180,E1 24685.291,E2 24685.291} C_VEL
LIN {X 0,Y 552.312,Z 605.435,A -85,B 0,C 180,E1 24681.896,E2 24681.896} C_VEL
LIN {X 0,Y 552.342,Z 605.433,A -85,B 0,C 180,E1 24678.578,E2 24678.578} C_VEL
LIN {X 0,Y 552.296,Z 605.435,A -85,B 0,C 180,E1 24675.326,E2 24675.326} C_VEL
LIN {X 0,Y 552.334,Z 605.437,A -85,B 0,C 180,E1 24672.015,E2 24672.015} C_VEL
LIN {X 0,Y 552.305,Z 605.435,A -85,B 0,C 180,E1 24668.747,E2 24668.747} C_VEL
LIN {X 0,Y 552.324,Z 605.614,A -85,B 0,C 180,E1 24665.532,E2 24665.532} C_VEL
LIN {X 0,Y 554.084,Z 613.683,A -85,B 0,C 180,E1 24664.554,E2 24664.554} C_VEL
LIN {X 0,Y 554.027,Z 640.651,A -85,B 0,C 180,E1 24661.551,E2 24661.551} C_VEL
LIN {X 0,Y 553.677,Z 670.244,A -85,B 0,C 180,E1 24658.137,E2 24658.137} C_VEL
LIN {X 0,Y 553.195,Z 693.452,A -85,B 0,C 180,E1 24655.373,E2 24655.373} C_VEL
LIN {X 0,Y 554.185,Z 701.18,A -85,B 0,C 180,E1 24655.223,E2 24655.223} C_VEL
LIN {X 0,Y 553.719,Z 832.88,A -85,B 0,C 180,E1 24653.464,E2 24653.464} C_VEL
LIN {X 0,Y 553.547,Z 849.962,A -85,B 0,C 180,E1 24653.026,E2 24653.026} C_VEL
LIN {X 0,Y 553.315,Z 865.503,A -85,B 0,C 180,E1 24652.42,E2 24652.42} C_VEL
LIN {X 0,Y 553.051,Z 880.498,A -85,B 0,C 180,E1 24651.631,E2 24651.631} C_VEL
LIN {X 0,Y 552.838,Z 891.396,A -85,B 0,C 180,E1 24650.908,E2 24650.908} C_VEL
LIN {X 0,Y 551.742,Z 897.714,A -85,B 0,C 180,E1 24650.452,E2 24650.452} C_VEL
LIN {X 0,Y 547.13,Z 908.629,A -85,B 0,C 180,E1 24649.57,E2 24649.57} C_VEL
LIN {X 0,Y 544.828,Z 914.894,A -85,B 0,C 180,E1 24648.949,E2 24648.949} C_VEL
LIN {X 0,Y 544.413,Z 917.883,A -85,B 0,C 180,E1 24648.606,E2 24648.606} C_VEL
LIN {X 0,Y 544.201,Z 928.797,A -85,B 0,C 180,E1 24647.155,E2 24647.155} C_VEL
LIN {X 0,Y 544.058,Z 937.741,A -85,B 0,C 180,E1 24645.635,E2 24645.635} C_VEL
LIN {X 0,Y 543.977,Z 944.756,A -85,B 0,C 180,E1 24644.105,E2 24644.105} C_VEL
LIN {X 0,Y 543.932,Z 950.296,A -85,B 0,C 180,E1 24642.454,E2 24642.454} C_VEL
LIN {X 0,Y 543.917,Z 954.072,A -85,B 0,C 180,E1 24640.789,E2 24640.789} C_VEL
LIN {X 0,Y 543.916,Z 956.076,A -85,B 0,C 180,E1 24639.107,E2 24639.107} C_VEL
LIN {X 0,Y 543.916,Z 956.378,A -85,B 0,C 180,E1 24637.341,E2 24637.341} C_VEL
LIN {X 0,Y 543.916,Z 954.924,A -85,B 0,C 180,E1 24635.684,E2 24635.684} C_VEL
LIN {X 0,Y 543.926,Z 951.583,A -85,B 0,C 180,E1 24633.938,E2 24633.938} C_VEL
LIN {X 0,Y 543.958,Z 946.558,A -85,B 0,C 180,E1 24632.287,E2 24632.287} C_VEL
LIN {X 0,Y 544.039,Z 939.472,A -85,B 0,C 180,E1 24630.613,E2 24630.613} C_VEL
LIN {X 0,Y 544.16,Z 931.018,A -85,B 0,C 180,E1 24629.103,E2 24629.103} C_VEL
LIN {X 0,Y 544.354,Z 920.857,A -85,B 0,C 180,E1 24627.664,E2 24627.664} C_VEL
LIN {X 0,Y 544.605,Z 908.919,A -85,B 0,C 180,E1 24626.327,E2 24626.327} C_VEL
LIN {X 0,Y 544.89,Z 896.465,A -85,B 0,C 180,E1 24625.202,E2 24625.202} C_VEL
LIN {X 0,Y 545.215,Z 882.533,A -85,B 0,C 180,E1 24624.196,E2 24624.196} C_VEL
LIN {X 0,Y 545.517,Z 868.309,A -85,B 0,C 180,E1 24623.398,E2 24623.398} C_VEL
LIN {X 0,Y 545.788,Z 852.892,A -85,B 0,C 180,E1 24622.757,E2 24622.757} C_VEL
LIN {X 0,Y 545.984,Z 836.883,A -85,B 0,C 180,E1 24622.303,E2 24622.303} C_VEL
LIN {X 0,Y 546.09,Z 813.855,A -85,B 0,C 180,E1 24621.942,E2 24621.942} C_VEL
LIN {X 0,Y 546.337,Z 699.217,A -85,B 0,C 180,E1 24620.403,E2 24620.403} C_VEL
LIN {X 0,Y 545.461,Z 693.735,A -85,B 0,C 180,E1 24620.262,E2 24620.262} C_VEL
LIN {X 0,Y 545.989,Z 665.408,A -85,B 0,C 180,E1 24616.916,E2 24616.916} C_VEL
LIN {X 0,Y 546.398,Z 638.516,A -85,B 0,C 180,E1 24613.766,E2 24613.766} C_VEL
LIN {X 0,Y 546.514,Z 615.682,A -85,B 0,C 180,E1 24611.126,E2 24611.126} C_VEL
LIN {X 0,Y 544.416,Z 606.545,A -85,B 0,C 180,E1 24609.926,E2 24609.926} C_VEL
LIN {X 0,Y 544.332,Z 606.413,A -85,B 0,C 180,E1 24606.785,E2 24606.785} C_VEL
LIN {X 0,Y 544.4,Z 606.419,A -85,B 0,C 180,E1 24603.505,E2 24603.505} C_VEL
LIN {X 0,Y 544.342,Z 606.424,A -85,B 0,C 180,E1 24600.31,E2 24600.31} C_VEL
LIN {X 0,Y 544.376,Z 606.421,A -85,B 0,C 180,E1 24596.98,E2 24596.98} C_VEL
LIN {X 0,Y 544.356,Z 606.415,A -85,B 0,C 180,E1 24593.834,E2 24593.834} C_VEL
LIN {X 0,Y 544.355,Z 606.417,A -85,B 0,C 180,E1 24590.426,E2 24590.426} C_VEL
LIN {X 0,Y 544.396,Z 606.423,A -85,B 0,C 180,E1 24587.2,E2 24587.2} C_VEL
LIN {X 0,Y 544.352,Z 606.427,A -85,B 0,C 180,E1 24583.923,E2 24583.923} C_VEL
LIN {X 0,Y 544.394,Z 606.693,A -85,B 0,C 180,E1 24581.505,E2 24581.505} C_VEL
LIN {X 0,Y 547.326,Z 618.661,A -85,B 0,C 180,E1 24579.782,E2 24579.782} C_VEL
LIN {X 0,Y 546.539,Z 645.963,A -85,B 0,C 180,E1 24576.408,E2 24576.408} C_VEL
LIN {X 0,Y 545.86,Z 673.576,A -85,B 0,C 180,E1 24573.045,E2 24573.045} C_VEL
LIN {X 0,Y 545.473,Z 692.835,A -85,B 0,C 180,E1 24570.749,E2 24570.749} C_VEL
LIN {X 0,Y 546.789,Z 702.068,A -85,B 0,C 180,E1 24570.544,E2 24570.544} C_VEL
LIN {X 0,Y 546.163,Z 833.513,A -85,B 0,C 180,E1 24568.732,E2 24568.732} C_VEL
LIN {X 0,Y 545.961,Z 850.348,A -85,B 0,C 180,E1 24568.288,E2 24568.288} C_VEL
LIN {X 0,Y 545.686,Z 865.442,A -85,B 0,C 180,E1 24567.69,E2 24567.69} C_VEL
LIN {X 0,Y 545.352,Z 880.119,A -85,B 0,C 180,E1 24566.9,E2 24566.9} C_VEL
LIN {X 0,Y 544.999,Z 893.825,A -85,B 0,C 180,E1 24565.95,E2 24565.95} C_VEL
LIN {X 0,Y 544.661,Z 906.949,A -85,B 0,C 180,E1 24564.787,E2 24564.787} C_VEL
LIN {X 0,Y 544.389,Z 919.107,A -85,B 0,C 180,E1 24563.462,E2 24563.462} C_VEL
LIN {X 0,Y 544.187,Z 929.6,A -85,B 0,C 180,E1 24562.028,E2 24562.028} C_VEL
LIN {X 0,Y 544.055,Z 938.021,A -85,B 0,C 180,E1 24560.586,E2 24560.586} C_VEL
LIN {X 0,Y 543.97,Z 945.236,A -85,B 0,C 180,E1 24558.974,E2 24558.974} C_VEL
LIN {X 0,Y 543.934,Z 950.551,A -85,B 0,C 180,E1 24557.365,E2 24557.365} C_VEL
LIN {X 0,Y 543.917,Z 954.155,A -85,B 0,C 180,E1 24555.74,E2 24555.74} C_VEL
LIN {X 0,Y 543.914,Z 956.145,A -85,B 0,C 180,E1 24553.994,E2 24553.994} C_VEL
LIN {X 0,Y 543.914,Z 956.343,A -85,B 0,C 180,E1 24552.233,E2 24552.233} C_VEL
LIN {X 0,Y 543.917,Z 954.755,A -85,B 0,C 180,E1 24550.566,E2 24550.566} C_VEL
LIN {X 0,Y 543.931,Z 951.433,A -85,B 0,C 180,E1 24548.882,E2 24548.882} C_VEL
LIN {X 0,Y 543.96,Z 946.606,A -85,B 0,C 180,E1 24547.294,E2 24547.294} C_VEL
LIN {X 0,Y 544.032,Z 939.817,A -85,B 0,C 180,E1 24545.69,E2 24545.69} C_VEL
LIN {X 0,Y 544.154,Z 931.553,A -85,B 0,C 180,E1 24544.185,E2 24544.185} C_VEL
LIN {X 0,Y 544.338,Z 921.517,A -85,B 0,C 180,E1 24542.752,E2 24542.752} C_VEL
LIN {X 0,Y 544.61,Z 909.266,A -85,B 0,C 180,E1 24541.351,E2 24541.351} C_VEL
LIN {X 0,Y 544.937,Z 896.602,A -85,B 0,C 180,E1 24540.183,E2 24540.183} C_VEL
LIN {X 0,Y 545.301,Z 882.821,A -85,B 0,C 180,E1 24539.171,E2 24539.171} C_VEL
LIN {X 0,Y 545.629,Z 868.537,A -85,B 0,C 180,E1 24538.362,E2 24538.362} C_VEL
LIN {X 0,Y 545.946,Z 852.892,A -85,B 0,C 180,E1 24537.701,E2 24537.701} C_VEL
LIN {X 0,Y 546.162,Z 837.095,A -85,B 0,C 180,E1 24537.247,E2 24537.247} C_VEL
LIN {X 0,Y 546.317,Z 814.009,A -85,B 0,C 180,E1 24536.876,E2 24536.876} C_VEL
LIN {X 0,Y 546.645,Z 699.161,A -85,B 0,C 180,E1 24535.303,E2 24535.303} C_VEL
LIN {X 0,Y 545.488,Z 692.759,A -85,B 0,C 180,E1 24535.135,E2 24535.135} C_VEL
LIN {X 0,Y 546.143,Z 664.782,A -85,B 0,C 180,E1 24531.758,E2 24531.758} C_VEL
LIN {X 0,Y 546.894,Z 637.607,A -85,B 0,C 180,E1 24528.421,E2 24528.421} C_VEL
LIN {X 0,Y 547.401,Z 617.762,A -85,B 0,C 180,E1 24525.944,E2 24525.944} C_VEL
LIN {X 0,Y 544.405,Z 606.517,A -85,B 0,C 180,E1 24524.252,E2 24524.252} C_VEL
LIN {X 0,Y 544.405,Z 606.425,A -85,B 0,C 180,E1 24520.828,E2 24520.828} C_VEL
LIN {X 0,Y 544.393,Z 606.42,A -85,B 0,C 180,E1 24517.44,E2 24517.44} C_VEL
LIN {X 0,Y 544.388,Z 606.421,A -85,B 0,C 180,E1 24514.069,E2 24514.069} C_VEL
LIN {X 0,Y 544.389,Z 606.421,A -85,B 0,C 180,E1 24510.704,E2 24510.704} C_VEL
LIN {X 0,Y 544.397,Z 606.418,A -85,B 0,C 180,E1 24507.333,E2 24507.333} C_VEL
LIN {X 0,Y 544.391,Z 606.423,A -85,B 0,C 180,E1 24503.833,E2 24503.833} C_VEL
LIN {X 0,Y 544.39,Z 606.42,A -85,B 0,C 180,E1 24500.497,E2 24500.497} C_VEL
LIN {X 0,Y 544.388,Z 606.419,A -85,B 0,C 180,E1 24497.09,E2 24497.09} C_VEL
LIN {X 0,Y 544.399,Z 606.423,A -85,B 0,C 180,E1 24493.597,E2 24493.597} C_VEL
LIN {X 0,Y 544.393,Z 606.415,A -85,B 0,C 180,E1 24490.156,E2 24490.156} C_VEL
LIN {X 0,Y 544.381,Z 606.419,A -85,B 0,C 180,E1 24486.857,E2 24486.857} C_VEL
LIN {X 0,Y 544.397,Z 606.422,A -85,B 0,C 180,E1 24483.475,E2 24483.475} C_VEL
LIN {X 0,Y 544.401,Z 606.412,A -85,B 0,C 180,E1 24480,E2 24480} C_VEL
LIN {X 0,Y 544.381,Z 606.417,A -85,B 0,C 180,E1 24476.631,E2 24476.631} C_VEL
LIN {X 0,Y 544.394,Z 606.42,A -85,B 0,C 180,E1 24473.25,E2 24473.25} C_VEL
LIN {X 0,Y 544.383,Z 606.416,A -85,B 0,C 180,E1 24469.885,E2 24469.885} C_VEL
LIN {X 0,Y 544.392,Z 606.419,A -85,B 0,C 180,E1 24466.403,E2 24466.403} C_VEL
LIN {X 0,Y 544.398,Z 606.419,A -85,B 0,C 180,E1 24463.021,E2 24463.021} C_VEL
LIN {X 0,Y 544.376,Z 606.421,A -85,B 0,C 180,E1 24459.688,E2 24459.688} C_VEL
LIN {X 0,Y 544.398,Z 606.418,A -85,B 0,C 180,E1 24456.398,E2 24456.398} C_VEL
LIN {X 0,Y 544.387,Z 606.415,A -85,B 0,C 180,E1 24453.022,E2 24453.022} C_VEL
LIN {X 0,Y 544.38,Z 606.42,A -85,B 0,C 180,E1 24449.541,E2 24449.541} C_VEL
LIN {X 0,Y 544.397,Z 606.421,A -85,B 0,C 180,E1 24446.186,E2 24446.186} C_VEL
LIN {X 0,Y 544.373,Z 606.42,A -85,B 0,C 180,E1 24442.823,E2 24442.823} C_VEL
LIN {X 0,Y 544.4,Z 606.423,A -85,B 0,C 180,E1 24439.446,E2 24439.446} C_VEL
LIN {X 0,Y 544.401,Z 606.415,A -85,B 0,C 180,E1 24436.033,E2 24436.033} C_VEL
LIN {X 0,Y 544.37,Z 606.424,A -85,B 0,C 180,E1 24432.668,E2 24432.668} C_VEL
LIN {X 0,Y 544.4,Z 606.421,A -85,B 0,C 180,E1 24429.455,E2 24429.455} C_VEL
LIN {X 0,Y 544.37,Z 606.427,A -85,B 0,C 180,E1 24426.128,E2 24426.128} C_VEL
LIN {X 0,Y 544.4,Z 606.656,A -85,B 0,C 180,E1 24424.194,E2 24424.194} C_VEL
LIN {X 0,Y 550.282,Z 623.298,A -85,B 0,C 180,E1 24422.48,E2 24422.48} C_VEL
LIN {X 0,Y 549.106,Z 666.368,A -85,B 0,C 180,E1 24419.149,E2 24419.149} C_VEL
LIN {X 0,Y 548.012,Z 709.272,A -85,B 0,C 180,E1 24415.92,E2 24415.92} C_VEL
LIN {X 0,Y 549.515,Z 720.192,A -85,B 0,C 180,E1 24415.676,E2 24415.676} C_VEL
LIN {X 0,Y 548.308,Z 927.53,A -85,B 0,C 180,E1 24412.788,E2 24412.788} C_VEL
LIN {X 0,Y 547.988,Z 946.963,A -85,B 0,C 180,E1 24412.317,E2 24412.317} C_VEL
LIN {X 0,Y 547.561,Z 965.939,A -85,B 0,C 180,E1 24411.652,E2 24411.652} C_VEL
LIN {X 0,Y 547.074,Z 983.811,A -85,B 0,C 180,E1 24410.822,E2 24410.822} C_VEL
LIN {X 0,Y 546.56,Z 1000.711,A -85,B 0,C 180,E1 24409.837,E2 24409.837} C_VEL
LIN {X 0,Y 546.018,Z 1017.51,A -85,B 0,C 180,E1 24408.631,E2 24408.631} C_VEL
LIN {X 0,Y 545.501,Z 1033.103,A -85,B 0,C 180,E1 24407.273,E2 24407.273} C_VEL
LIN {X 0,Y 545.069,Z 1046.685,A -85,B 0,C 180,E1 24405.862,E2 24405.862} C_VEL
LIN {X 0,Y 544.683,Z 1059.754,A -85,B 0,C 180,E1 24404.239,E2 24404.239} C_VEL
LIN {X 0,Y 544.384,Z 1071.298,A -85,B 0,C 180,E1 24402.517,E2 24402.517} C_VEL
LIN {X 0,Y 544.175,Z 1081.335,A -85,B 0,C 180,E1 24400.694,E2 24400.694} C_VEL
LIN {X 0,Y 544.04,Z 1089.433,A -85,B 0,C 180,E1 24398.88,E2 24398.88} C_VEL
LIN {X 0,Y 543.958,Z 1096.129,A -85,B 0,C 180,E1 24396.968,E2 24396.968} C_VEL
LIN {X 0,Y 543.923,Z 1101.297,A -85,B 0,C 180,E1 24394.956,E2 24394.956} C_VEL
LIN {X 0,Y 543.908,Z 1104.659,A -85,B 0,C 180,E1 24392.95,E2 24392.95} C_VEL
LIN {X 0,Y 543.909,Z 1106.304,A -85,B 0,C 180,E1 24390.948,E2 24390.948} C_VEL
LIN {X 0,Y 543.906,Z 1106.264,A -85,B 0,C 180,E1 24388.946,E2 24388.946} C_VEL
LIN {X 0,Y 543.912,Z 1104.538,A -85,B 0,C 180,E1 24386.944,E2 24386.944} C_VEL
LIN {X 0,Y 543.922,Z 1101.086,A -85,B 0,C 180,E1 24384.938,E2 24384.938} C_VEL
LIN {X 0,Y 543.964,Z 1095.818,A -85,B 0,C 180,E1 24382.926,E2 24382.926} C_VEL
LIN {X 0,Y 544.045,Z 1088.592,A -85,B 0,C 180,E1 24380.906,E2 24380.906} C_VEL
LIN {X 0,Y 544.205,Z 1079.734,A -85,B 0,C 180,E1 24378.984,E2 24378.984} C_VEL
LIN {X 0,Y 544.434,Z 1069.309,A -85,B 0,C 180,E1 24377.16,E2 24377.16} C_VEL
LIN {X 0,Y 544.754,Z 1057.323,A -85,B 0,C 180,E1 24375.436,E2 24375.436} C_VEL
LIN {X 0,Y 545.151,Z 1044.233,A -85,B 0,C 180,E1 24373.867,E2 24373.867} C_VEL
LIN {X 0,Y 545.622,Z 1029.588,A -85,B 0,C 180,E1 24372.4,E2 24372.4} C_VEL
LIN {X 0,Y 546.14,Z 1013.897,A -85,B 0,C 180,E1 24371.092,E2 24371.092} C_VEL
LIN {X 0,Y 546.675,Z 996.927,A -85,B 0,C 180,E1 24369.928,E2 24369.928} C_VEL
LIN {X 0,Y 547.194,Z 979.431,A -85,B 0,C 180,E1 24368.958,E2 24368.958} C_VEL
LIN {X 0,Y 547.66,Z 961.125,A -85,B 0,C 180,E1 24368.162,E2 24368.162} C_VEL
LIN {X 0,Y 548.056,Z 941.786,A -85,B 0,C 180,E1 24367.54,E2 24367.54} C_VEL
LIN {X 0,Y 548.354,Z 922.013,A -85,B 0,C 180,E1 24367.119,E2 24367.119} C_VEL
LIN {X 0,Y 549.356,Z 717.642,A -85,B 0,C 180,E1 24364.28,E2 24364.28} C_VEL
LIN {X 0,Y 548.023,Z 709.44,A -85,B 0,C 180,E1 24364.088,E2 24364.088} C_VEL
LIN {X 0,Y 549.076,Z 667.471,A -85,B 0,C 180,E1 24360.935,E2 24360.935} C_VEL
LIN {X 0,Y 550.267,Z 624.173,A -85,B 0,C 180,E1 24357.586,E2 24357.586} C_VEL
LIN {X 0,Y 549.782,Z 621.599,A -85,B 0,C 180,E1 24357.355,E2 24357.355} C_VEL
LIN {X 0,Y 544.407,Z 606.673,A -85,B 0,C 180,E1 24355.797,E2 24355.797} C_VEL
LIN {X 0,Y 544.398,Z 606.425,A -85,B 0,C 180,E1 24352.68,E2 24352.68} C_VEL
LIN {X 0,Y 544.387,Z 606.424,A -85,B 0,C 180,E1 24349.306,E2 24349.306} C_VEL
LIN {X 0,Y 544.397,Z 606.416,A -85,B 0,C 180,E1 24345.886,E2 24345.886} C_VEL
LIN {X 0,Y 544.391,Z 606.423,A -85,B 0,C 180,E1 24342.523,E2 24342.523} C_VEL
LIN {X 0,Y 544.388,Z 606.423,A -85,B 0,C 180,E1 24339.184,E2 24339.184} C_VEL
LIN {X 0,Y 544.39,Z 606.419,A -85,B 0,C 180,E1 24335.866,E2 24335.866} C_VEL
LIN {X 0,Y 544.393,Z 606.426,A -85,B 0,C 180,E1 24332.432,E2 24332.432} C_VEL
LIN {X 0,Y 544.399,Z 606.42,A -85,B 0,C 180,E1 24329.004,E2 24329.004} C_VEL
LIN {X 0,Y 544.372,Z 606.422,A -85,B 0,C 180,E1 24325.688,E2 24325.688} C_VEL
LIN {X 0,Y 544.4,Z 606.426,A -85,B 0,C 180,E1 24322.345,E2 24322.345} C_VEL
LIN {X 0,Y 544.393,Z 606.419,A -85,B 0,C 180,E1 24318.936,E2 24318.936} C_VEL
LIN {X 0,Y 544.358,Z 606.425,A -85,B 0,C 180,E1 24315.555,E2 24315.555} C_VEL
LIN {X 0,Y 544.406,Z 606.424,A -85,B 0,C 180,E1 24312.29,E2 24312.29} C_VEL
LIN {X 0,Y 544.353,Z 606.426,A -85,B 0,C 180,E1 24308.982,E2 24308.982} C_VEL
LIN {X 0,Y 544.411,Z 606.623,A -85,B 0,C 180,E1 24305.771,E2 24305.771} C_VEL
LIN {X 0,Y 546.419,Z 616.238,A -85,B 0,C 180,E1 24304.618,E2 24304.618} C_VEL
LIN {X 0,Y 546.372,Z 641.741,A -85,B 0,C 180,E1 24301.783,E2 24301.783} C_VEL
LIN {X 0,Y 546.056,Z 670.011,A -85,B 0,C 180,E1 24298.531,E2 24298.531} C_VEL
LIN {X 0,Y 545.607,Z 694.754,A -85,B 0,C 180,E1 24295.612,E2 24295.612} C_VEL
LIN {X 0,Y 546.549,Z 702.229,A -85,B 0,C 180,E1 24295.46,E2 24295.46} C_VEL
LIN {X 0,Y 546.002,Z 833.81,A -85,B 0,C 180,E1 24293.672,E2 24293.672} C_VEL
LIN {X 0,Y 545.826,Z 850.7,A -85,B 0,C 180,E1 24293.231,E2 24293.231} C_VEL
LIN {X 0,Y 545.573,Z 865.881,A -85,B 0,C 180,E1 24292.629,E2 24292.629} C_VEL
LIN {X 0,Y 545.263,Z 880.784,A -85,B 0,C 180,E1 24291.83,E2 24291.83} C_VEL
LIN {X 0,Y 544.93,Z 894.482,A -85,B 0,C 180,E1 24290.868,E2 24290.868} C_VEL
LIN {X 0,Y 544.644,Z 907.414,A -85,B 0,C 180,E1 24289.736,E2 24289.736} C_VEL
LIN {X 0,Y 544.413,Z 917.883,A -85,B 0,C 180,E1 24288.606,E2 24288.606} C_VEL
LIN {X 0,Y 543.321,Z 922.932,A -85,B 0,C 180,E1 24287.993,E2 24287.993} C_VEL
LIN {X 0,Y 538.388,Z 932.092,A -85,B 0,C 180,E1 24286.754,E2 24286.754} C_VEL
LIN {X 0,Y 536.318,Z 936.783,A -85,B 0,C 180,E1 24285.975,E2 24285.975} C_VEL
LIN {X 0,Y 536.086,Z 938.367,A -85,B 0,C 180,E1 24285.664,E2 24285.664} C_VEL
LIN {X 0,Y 535.977,Z 945.607,A -85,B 0,C 180,E1 24283.973,E2 24283.973} C_VEL
LIN {X 0,Y 535.931,Z 951.217,A -85,B 0,C 180,E1 24282.183,E2 24282.183} C_VEL
LIN {X 0,Y 535.917,Z 954.691,A -85,B 0,C 180,E1 24280.422,E2 24280.422} C_VEL
LIN {X 0,Y 535.914,Z 956.353,A -85,B 0,C 180,E1 24278.665,E2 24278.665} C_VEL
LIN {X 0,Y 535.916,Z 956.143,A -85,B 0,C 180,E1 24276.896,E2 24276.896} C_VEL
LIN {X 0,Y 535.919,Z 954.243,A -85,B 0,C 180,E1 24275.179,E2 24275.179} C_VEL
LIN {X 0,Y 535.933,Z 950.651,A -85,B 0,C 180,E1 24273.52,E2 24273.52} C_VEL
LIN {X 0,Y 535.98,Z 945.231,A -85,B 0,C 180,E1 24271.838,E2 24271.838} C_VEL
LIN {X 0,Y 536.096,Z 937.764,A -85,B 0,C 180,E1 24270.134,E2 24270.134} C_VEL
LIN {X 0,Y 536.279,Z 929.33,A -85,B 0,C 180,E1 24268.641,E2 24268.641} C_VEL
LIN {X 0,Y 536.544,Z 918.834,A -85,B 0,C 180,E1 24267.188,E2 24267.188} C_VEL
LIN {X 0,Y 536.848,Z 907.936,A -85,B 0,C 180,E1 24265.976,E2 24265.976} C_VEL
LIN {X 0,Y 537.195,Z 894.595,A -85,B 0,C 180,E1 24264.795,E2 24264.795} C_VEL
LIN {X 0,Y 537.547,Z 880.708,A -85,B 0,C 180,E1 24263.829,E2 24263.829} C_VEL
LIN {X 0,Y 537.872,Z 865.912,A -85,B 0,C 180,E1 24263.039,E2 24263.039} C_VEL
LIN {X 0,Y 538.13,Z 850.104,A -85,B 0,C 180,E1 24262.424,E2 24262.424} C_VEL
LIN {X 0,Y 538.302,Z 833.504,A -85,B 0,C 180,E1 24262,E2 24262} C_VEL
LIN {X 0,Y 538.702,Z 700.124,A -85,B 0,C 180,E1 24260.154,E2 24260.154} C_VEL
LIN {X 0,Y 537.808,Z 694.726,A -85,B 0,C 180,E1 24260.014,E2 24260.014} C_VEL
LIN {X 0,Y 538.385,Z 664.605,A -85,B 0,C 180,E1 24256.449,E2 24256.449} C_VEL
LIN {X 0,Y 538.769,Z 636.511,A -85,B 0,C 180,E1 24253.169,E2 24253.169} C_VEL
LIN {X 0,Y 538.795,Z 617.508,A -85,B 0,C 180,E1 24250.949,E2 24250.949} C_VEL
LIN {X 0,Y 536.467,Z 607.554,A -85,B 0,C 180,E1 24249.655,E2 24249.655} C_VEL
LIN {X 0,Y 536.398,Z 607.402,A -85,B 0,C 180,E1 24246.486,E2 24246.486} C_VEL
LIN {X 0,Y 536.42,Z 607.411,A -85,B 0,C 180,E1 24243.103,E2 24243.103} C_VEL
LIN {X 0,Y 536.421,Z 607.415,A -85,B 0,C 180,E1 24239.97,E2 24239.97} C_VEL
LIN {X 0,Y 536.407,Z 607.411,A -85,B 0,C 180,E1 24236.575,E2 24236.575} C_VEL
LIN {X 0,Y 536.465,Z 607.406,A -85,B 0,C 180,E1 24233.274,E2 24233.274} C_VEL
LIN {X 0,Y 536.408,Z 607.407,A -85,B 0,C 180,E1 24229.945,E2 24229.945} C_VEL
LIN {X 0,Y 536.443,Z 607.403,A -85,B 0,C 180,E1 24226.569,E2 24226.569} C_VEL
LIN {X 0,Y 536.43,Z 607.415,A -85,B 0,C 180,E1 24223.352,E2 24223.352} C_VEL
LIN {X 0,Y 536.456,Z 607.713,A -85,B 0,C 180,E1 24221.876,E2 24221.876} C_VEL
LIN {X 0,Y 539.813,Z 620.326,A -85,B 0,C 180,E1 24220.027,E2 24220.027} C_VEL
LIN {X 0,Y 538.978,Z 646.83,A -85,B 0,C 180,E1 24216.712,E2 24216.712} C_VEL
LIN {X 0,Y 538.203,Z 674.43,A -85,B 0,C 180,E1 24213.302,E2 24213.302} C_VEL
LIN {X 0,Y 537.802,Z 693.087,A -85,B 0,C 180,E1 24211.066,E2 24211.066} C_VEL
LIN {X 0,Y 539.348,Z 702.808,A -85,B 0,C 180,E1 24210.847,E2 24210.847} C_VEL
LIN {X 0,Y 538.633,Z 834.145,A -85,B 0,C 180,E1 24209.01,E2 24209.01} C_VEL
LIN {X 0,Y 538.414,Z 851.006,A -85,B 0,C 180,E1 24208.56,E2 24208.56} C_VEL
LIN {X 0,Y 538.129,Z 865.683,A -85,B 0,C 180,E1 24207.977,E2 24207.977} C_VEL
LIN {X 0,Y 537.756,Z 880.496,A -85,B 0,C 180,E1 24207.176,E2 24207.176} C_VEL
LIN {X 0,Y 537.358,Z 894.328,A -85,B 0,C 180,E1 24206.213,E2 24206.213} C_VEL
LIN {X 0,Y 536.982,Z 907.027,A -85,B 0,C 180,E1 24205.087,E2 24205.087} C_VEL
LIN {X 0,Y 536.633,Z 918.719,A -85,B 0,C 180,E1 24203.796,E2 24203.796} C_VEL
LIN {X 0,Y 536.338,Z 928.853,A -85,B 0,C 180,E1 24202.394,E2 24202.394} C_VEL
LIN {X 0,Y 536.118,Z 938.084,A -85,B 0,C 180,E1 24200.771,E2 24200.771} C_VEL
LIN {X 0,Y 535.997,Z 944.726,A -85,B 0,C 180,E1 24199.249,E2 24199.249} C_VEL
LIN {X 0,Y 535.939,Z 950.383,A -85,B 0,C 180,E1 24197.502,E2 24197.502} C_VEL
LIN {X 0,Y 535.918,Z 954.211,A -85,B 0,C 180,E1 24195.743,E2 24195.743} C_VEL
LIN {X 0,Y 535.914,Z 956.169,A -85,B 0,C 180,E1 24193.971,E2 24193.971} C_VEL
LIN {X 0,Y 535.914,Z 956.366,A -85,B 0,C 180,E1 24192.296,E2 24192.296} C_VEL
LIN {X 0,Y 535.917,Z 954.865,A -85,B 0,C 180,E1 24190.604,E2 24190.604} C_VEL
LIN {X 0,Y 535.932,Z 951.35,A -85,B 0,C 180,E1 24188.781,E2 24188.781} C_VEL
LIN {X 0,Y 535.98,Z 946.17,A -85,B 0,C 180,E1 24187.053,E2 24187.053} C_VEL
LIN {X 0,Y 536.091,Z 939.482,A -85,B 0,C 180,E1 24185.423,E2 24185.423} C_VEL
LIN {X 0,Y 536.287,Z 931.306,A -85,B 0,C 180,E1 24183.896,E2 24183.896} C_VEL
LIN {X 0,Y 536.573,Z 921.177,A -85,B 0,C 180,E1 24182.416,E2 24182.416} C_VEL
LIN {X 0,Y 536.91,Z 910.528,A -85,B 0,C 180,E1 24181.163,E2 24181.163} C_VEL
LIN {X 0,Y 537.291,Z 897.713,A -85,B 0,C 180,E1 24179.961,E2 24179.961} C_VEL
LIN {X 0,Y 537.7,Z 883.978,A -85,B 0,C 180,E1 24178.936,E2 24178.936} C_VEL
LIN {X 0,Y 538.079,Z 869.251,A -85,B 0,C 180,E1 24178.092,E2 24178.092} C_VEL
LIN {X 0,Y 538.428,Z 853.433,A -85,B 0,C 180,E1 24177.417,E2 24177.417} C_VEL
LIN {X 0,Y 538.654,Z 837.578,A -85,B 0,C 180,E1 24176.959,E2 24176.959} C_VEL
LIN {X 0,Y 538.821,Z 814.29,A -85,B 0,C 180,E1 24176.583,E2 24176.583} C_VEL
LIN {X 0,Y 539.239,Z 700.2,A -85,B 0,C 180,E1 24174.995,E2 24174.995} C_VEL
LIN {X 0,Y 537.83,Z 693.024,A -85,B 0,C 180,E1 24174.809,E2 24174.809} C_VEL
LIN {X 0,Y 538.541,Z 665.604,A -85,B 0,C 180,E1 24171.471,E2 24171.471} C_VEL
LIN {X 0,Y 539.367,Z 638.811,A -85,B 0,C 180,E1 24168.137,E2 24168.137} C_VEL
LIN {X 0,Y 539.882,Z 620.214,A -85,B 0,C 180,E1 24165.785,E2 24165.785} C_VEL
LIN {X 0,Y 536.477,Z 607.539,A -85,B 0,C 180,E1 24163.866,E2 24163.866} C_VEL
LIN {X 0,Y 536.452,Z 607.412,A -85,B 0,C 180,E1 24160.438,E2 24160.438} C_VEL
LIN {X 0,Y 536.449,Z 607.413,A -85,B 0,C 180,E1 24157.087,E2 24157.087} C_VEL
LIN {X 0,Y 536.454,Z 607.407,A -85,B 0,C 180,E1 24153.74,E2 24153.74} C_VEL
LIN {X 0,Y 536.46,Z 607.414,A -85,B 0,C 180,E1 24150.214,E2 24150.214} C_VEL
LIN {X 0,Y 536.452,Z 607.41,A -85,B 0,C 180,E1 24146.776,E2 24146.776} C_VEL
LIN {X 0,Y 536.449,Z 607.408,A -85,B 0,C 180,E1 24143.391,E2 24143.391} C_VEL
LIN {X 0,Y 536.462,Z 607.414,A -85,B 0,C 180,E1 24139.943,E2 24139.943} C_VEL
LIN {X 0,Y 536.455,Z 607.408,A -85,B 0,C 180,E1 24136.458,E2 24136.458} C_VEL
LIN {X 0,Y 536.444,Z 607.411,A -85,B 0,C 180,E1 24133.144,E2 24133.144} C_VEL
LIN {X 0,Y 536.455,Z 607.407,A -85,B 0,C 180,E1 24129.765,E2 24129.765} C_VEL
LIN {X 0,Y 536.464,Z 607.403,A -85,B 0,C 180,E1 24126.313,E2 24126.313} C_VEL
LIN {X 0,Y 536.446,Z 607.411,A -85,B 0,C 180,E1 24122.885,E2 24122.885} C_VEL
LIN {X 0,Y 536.456,Z 607.404,A -85,B 0,C 180,E1 24119.573,E2 24119.573} C_VEL
LIN {X 0,Y 536.441,Z 607.402,A -85,B 0,C 180,E1 24116.26,E2 24116.26} C_VEL
LIN {X 0,Y 536.462,Z 607.413,A -85,B 0,C 180,E1 24112.827,E2 24112.827} C_VEL
LIN {X 0,Y 536.46,Z 607.404,A -85,B 0,C 180,E1 24109.367,E2 24109.367} C_VEL
LIN {X 0,Y 536.438,Z 607.405,A -85,B 0,C 180,E1 24105.978,E2 24105.978} C_VEL
LIN {X 0,Y 536.461,Z 607.413,A -85,B 0,C 180,E1 24102.605,E2 24102.605} C_VEL
LIN {X 0,Y 536.462,Z 607.406,A -85,B 0,C 180,E1 24099.146,E2 24099.146} C_VEL
LIN {X 0,Y 536.438,Z 607.412,A -85,B 0,C 180,E1 24095.675,E2 24095.675} C_VEL
LIN {X 0,Y 536.458,Z 607.407,A -85,B 0,C 180,E1 24092.29,E2 24092.29} C_VEL
LIN {X 0,Y 536.443,Z 607.403,A -85,B 0,C 180,E1 24088.916,E2 24088.916} C_VEL
LIN {X 0,Y 536.446,Z 607.41,A -85,B 0,C 180,E1 24085.469,E2 24085.469} C_VEL
LIN {X 0,Y 536.461,Z 607.408,A -85,B 0,C 180,E1 24082.035,E2 24082.035} C_VEL
LIN {X 0,Y 536.434,Z 607.41,A -85,B 0,C 180,E1 24078.69,E2 24078.69} C_VEL
LIN {X 0,Y 536.456,Z 607.416,A -85,B 0,C 180,E1 24075.209,E2 24075.209} C_VEL
LIN {X 0,Y 536.461,Z 607.408,A -85,B 0,C 180,E1 24071.796,E2 24071.796} C_VEL
LIN {X 0,Y 536.43,Z 607.413,A -85,B 0,C 180,E1 24068.479,E2 24068.479} C_VEL
LIN {X 0,Y 536.463,Z 607.404,A -85,B 0,C 180,E1 24065.094,E2 24065.094} C_VEL
LIN {X 0,Y 536.493,Z 607.752,A -85,B 0,C 180,E1 24064.605,E2 24064.605} C_VEL
LIN {X 0,Y 542.949,Z 626.01,A -85,B 0,C 180,E1 24062.693,E2 24062.693} C_VEL
LIN {X 0,Y 541.937,Z 663.305,A -85,B 0,C 180,E1 24059.816,E2 24059.816} C_VEL
LIN {X 0,Y 540.639,Z 707.719,A -85,B 0,C 180,E1 24056.409,E2 24056.409} C_VEL
LIN {X 0,Y 540.768,Z 710.408,A -85,B 0,C 180,E1 24056.267,E2 24056.267} C_VEL
LIN {X 0,Y 542.3,Z 721.351,A -85,B 0,C 180,E1 24056.026,E2 24056.026} C_VEL
LIN {X 0,Y 540.931,Z 927.53,A -85,B 0,C 180,E1 24053.117,E2 24053.117} C_VEL
LIN {X 0,Y 540.571,Z 946.885,A -85,B 0,C 180,E1 24052.643,E2 24052.643} C_VEL
LIN {X 0,Y 540.12,Z 964.797,A -85,B 0,C 180,E1 24052.016,E2 24052.016} C_VEL
LIN {X 0,Y 539.571,Z 982.788,A -85,B 0,C 180,E1 24051.183,E2 24051.183} C_VEL
LIN {X 0,Y 538.952,Z 1000.707,A -85,B 0,C 180,E1 24050.129,E2 24050.129} C_VEL
LIN {X 0,Y 538.34,Z 1017.461,A -85,B 0,C 180,E1 24048.911,E2 24048.911} C_VEL
LIN {X 0,Y 537.75,Z 1033.102,A -85,B 0,C 180,E1 24047.53,E2 24047.53} C_VEL
LIN {X 0,Y 537.255,Z 1046.684,A -85,B 0,C 180,E1 24046.099,E2 24046.099} C_VEL
LIN {X 0,Y 536.807,Z 1059.755,A -85,B 0,C 180,E1 24044.453,E2 24044.453} C_VEL
LIN {X 0,Y 536.46,Z 1071.299,A -85,B 0,C 180,E1 24042.705,E2 24042.705} C_VEL
LIN {X 0,Y 536.218,Z 1081.336,A -85,B 0,C 180,E1 24040.855,E2 24040.855} C_VEL
LIN {X 0,Y 536.057,Z 1089.433,A -85,B 0,C 180,E1 24039.014,E2 24039.014} C_VEL
LIN {X 0,Y 535.968,Z 1096.212,A -85,B 0,C 180,E1 24037.042,E2 24037.042} C_VEL
LIN {X 0,Y 535.923,Z 1101.296,A -85,B 0,C 180,E1 24035.03,E2 24035.03} C_VEL
LIN {X 0,Y 535.91,Z 1104.659,A -85,B 0,C 180,E1 24032.994,E2 24032.994} C_VEL
LIN {X 0,Y 535.909,Z 1106.304,A -85,B 0,C 180,E1 24030.962,E2 24030.962} C_VEL
LIN {X 0,Y 535.906,Z 1106.264,A -85,B 0,C 180,E1 24028.931,E2 24028.931} C_VEL
LIN {X 0,Y 535.913,Z 1104.538,A -85,B 0,C 180,E1 24026.898,E2 24026.898} C_VEL
LIN {X 0,Y 535.922,Z 1101.086,A -85,B 0,C 180,E1 24024.862,E2 24024.862} C_VEL
LIN {X 0,Y 535.974,Z 1095.818,A -85,B 0,C 180,E1 24022.82,E2 24022.82} C_VEL
LIN {X 0,Y 536.069,Z 1088.592,A -85,B 0,C 180,E1 24020.769,E2 24020.769} C_VEL
LIN {X 0,Y 536.253,Z 1079.733,A -85,B 0,C 180,E1 24018.819,E2 24018.819} C_VEL
LIN {X 0,Y 536.523,Z 1069.308,A -85,B 0,C 180,E1 24016.968,E2 24016.968} C_VEL
LIN {X 0,Y 536.889,Z 1057.322,A -85,B 0,C 180,E1 24015.218,E2 24015.218} C_VEL
LIN {X 0,Y 537.343,Z 1044.233,A -85,B 0,C 180,E1 24013.626,E2 24013.626} C_VEL
LIN {X 0,Y 537.882,Z 1029.589,A -85,B 0,C 180,E1 24012.138,E2 24012.138} C_VEL
LIN {X 0,Y 538.474,Z 1013.899,A -85,B 0,C 180,E1 24010.812,E2 24010.812} C_VEL
LIN {X 0,Y 539.068,Z 997.443,A -85,B 0,C 180,E1 24009.665,E2 24009.665} C_VEL
LIN {X 0,Y 539.639,Z 980.554,A -85,B 0,C 180,E1 24008.706,E2 24008.706} C_VEL
LIN {X 0,Y 540.165,Z 962.599,A -85,B 0,C 180,E1 24007.9,E2 24007.9} C_VEL
LIN {X 0,Y 540.618,Z 943.867,A -85,B 0,C 180,E1 24007.271,E2 24007.271} C_VEL
LIN {X 0,Y 540.961,Z 924.797,A -85,B 0,C 180,E1 24006.835,E2 24006.835} C_VEL
LIN {X 0,Y 542.155,Z 718.876,A -85,B 0,C 180,E1 24003.931,E2 24003.931} C_VEL
LIN {X 0,Y 540.627,Z 709.114,A -85,B 0,C 180,E1 24003.687,E2 24003.687} C_VEL
LIN {X 0,Y 541.885,Z 665.435,A -85,B 0,C 180,E1 24000.35,E2 24000.35} C_VEL
LIN {X 0,Y 543.001,Z 625.92,A -85,B 0,C 180,E1 23997.286,E2 23997.286} C_VEL
LIN {X 0,Y 536.488,Z 607.663,A -85,B 0,C 180,E1 23995.359,E2 23995.359} C_VEL
LIN {X 0,Y 536.447,Z 607.412,A -85,B 0,C 180,E1 23992.042,E2 23992.042} C_VEL
LIN {X 0,Y 536.458,Z 607.411,A -85,B 0,C 180,E1 23988.687,E2 23988.687} C_VEL
LIN {X 0,Y 536.449,Z 607.411,A -85,B 0,C 180,E1 23985.245,E2 23985.245} C_VEL
LIN {X 0,Y 536.46,Z 607.406,A -85,B 0,C 180,E1 23981.795,E2 23981.795} C_VEL
LIN {X 0,Y 536.447,Z 607.412,A -85,B 0,C 180,E1 23978.364,E2 23978.364} C_VEL
LIN {X 0,Y 536.454,Z 607.412,A -85,B 0,C 180,E1 23975.034,E2 23975.034} C_VEL
LIN {X 0,Y 536.453,Z 607.407,A -85,B 0,C 180,E1 23971.594,E2 23971.594} C_VEL
LIN {X 0,Y 536.442,Z 607.413,A -85,B 0,C 180,E1 23968.135,E2 23968.135} C_VEL
LIN {X 0,Y 536.462,Z 607.411,A -85,B 0,C 180,E1 23964.794,E2 23964.794} C_VEL
LIN {X 0,Y 536.432,Z 607.41,A -85,B 0,C 180,E1 23961.427,E2 23961.427} C_VEL
LIN {X 0,Y 536.445,Z 607.416,A -85,B 0,C 180,E1 23958.023,E2 23958.023} C_VEL
LIN {X 0,Y 536.461,Z 607.41,A -85,B 0,C 180,E1 23954.683,E2 23954.683} C_VEL
LIN {X 0,Y 536.414,Z 607.415,A -85,B 0,C 180,E1 23951.347,E2 23951.347} C_VEL
LIN {X 0,Y 536.467,Z 607.413,A -85,B 0,C 180,E1 23948.035,E2 23948.035} C_VEL
LIN {X 0,Y 536.503,Z 607.675,A -85,B 0,C 180,E1 23946.017,E2 23946.017} C_VEL
LIN {X 0,Y 538.771,Z 618.365,A -85,B 0,C 180,E1 23944.741,E2 23944.741} C_VEL
LIN {X 0,Y 538.731,Z 645.764,A -85,B 0,C 180,E1 23941.701,E2 23941.701} C_VEL
LIN {X 0,Y 538.373,Z 675.276,A -85,B 0,C 180,E1 23938.297,E2 23938.297} C_VEL
LIN {X 0,Y 538.066,Z 696.38,A -85,B 0,C 180,E1 23935.84,E2 23935.84} C_VEL
LIN {X 0,Y 538.925,Z 703.249,A -85,B 0,C 180,E1 23935.706,E2 23935.706} C_VEL
LIN {X 0,Y 538.294,Z 835.415,A -85,B 0,C 180,E1 23933.872,E2 23933.872} C_VEL
LIN {X 0,Y 538.122,Z 851.946,A -85,B 0,C 180,E1 23933.432,E2 23933.432} C_VEL
LIN {X 0,Y 537.881,Z 866.686,A -85,B 0,C 180,E1 23932.845,E2 23932.845} C_VEL
LIN {X 0,Y 537.555,Z 881.691,A -85,B 0,C 180,E1 23932.035,E2 23932.035} C_VEL
LIN {X 0,Y 537.203,Z 895.493,A -85,B 0,C 180,E1 23931.059,E2 23931.059} C_VEL
LIN {X 0,Y 536.866,Z 908.267,A -85,B 0,C 180,E1 23929.917,E2 23929.917} C_VEL
LIN {X 0,Y 536.531,Z 920.003,A -85,B 0,C 180,E1 23928.591,E2 23928.591} C_VEL
LIN {X 0,Y 536.272,Z 929.964,A -85,B 0,C 180,E1 23927.181,E2 23927.181} C_VEL
LIN {X 0,Y 536.086,Z 938.367,A -85,B 0,C 180,E1 23925.664,E2 23925.664} C_VEL
LIN {X 0,Y 535.053,Z 941.952,A -85,B 0,C 180,E1 23924.935,E2 23924.935} C_VEL
LIN {X 0,Y 530.245,Z 948.315,A -85,B 0,C 180,E1 23923.482,E2 23923.482} C_VEL
LIN {X 0,Y 528.163,Z 951.397,A -85,B 0,C 180,E1 23922.539,E2 23922.539} C_VEL
LIN {X 0,Y 528.005,Z 952.163,A -85,B 0,C 180,E1 23922.25,E2 23922.25} C_VEL
LIN {X 0,Y 527.964,Z 955.41,A -85,B 0,C 180,E1 23920.53,E2 23920.53} C_VEL
LIN {X 0,Y 527.949,Z 957.094,A -85,B 0,C 180,E1 23918.677,E2 23918.677} C_VEL
LIN {X 0,Y 527.95,Z 956.833,A -85,B 0,C 180,E1 23916.801,E2 23916.801} C_VEL
LIN {X 0,Y 527.966,Z 954.836,A -85,B 0,C 180,E1 23915.019,E2 23915.019} C_VEL
LIN {X 0,Y 528.011,Z 950.923,A -85,B 0,C 180,E1 23913.212,E2 23913.212} C_VEL
LIN {X 0,Y 528.104,Z 945.358,A -85,B 0,C 180,E1 23911.503,E2 23911.503} C_VEL
LIN {X 0,Y 528.248,Z 938.191,A -85,B 0,C 180,E1 23909.884,E2 23909.884} C_VEL
LIN {X 0,Y 528.466,Z 929.471,A -85,B 0,C 180,E1 23908.365,E2 23908.365} C_VEL
LIN {X 0,Y 528.771,Z 918.765,A -85,B 0,C 180,E1 23906.896,E2 23906.896} C_VEL
LIN {X 0,Y 529.107,Z 907.57,A -85,B 0,C 180,E1 23905.671,E2 23905.671} C_VEL
LIN {X 0,Y 529.461,Z 895.032,A -85,B 0,C 180,E1 23904.566,E2 23904.566} C_VEL
LIN {X 0,Y 529.83,Z 881.287,A -85,B 0,C 180,E1 23903.608,E2 23903.608} C_VEL
LIN {X 0,Y 530.161,Z 867.03,A -85,B 0,C 180,E1 23902.84,E2 23902.84} C_VEL
LIN {X 0,Y 530.434,Z 850.971,A -85,B 0,C 180,E1 23902.206,E2 23902.206} C_VEL
LIN {X 0,Y 530.599,Z 834.607,A -85,B 0,C 180,E1 23901.785,E2 23901.785} C_VEL
LIN {X 0,Y 531.1,Z 701.135,A -85,B 0,C 180,E1 23899.901,E2 23899.901} C_VEL
LIN {X 0,Y 530.174,Z 695.874,A -85,B 0,C 180,E1 23899.773,E2 23899.773} C_VEL
LIN {X 0,Y 530.723,Z 666.073,A -85,B 0,C 180,E1 23896.258,E2 23896.258} C_VEL
LIN {X 0,Y 531.144,Z 638.703,A -85,B 0,C 180,E1 23893.039,E2 23893.039} C_VEL
LIN {X 0,Y 531.166,Z 619.704,A -85,B 0,C 180,E1 23890.824,E2 23890.824} C_VEL
LIN {X 0,Y 528.496,Z 608.554,A -85,B 0,C 180,E1 23889.365,E2 23889.365} C_VEL
LIN {X 0,Y 528.47,Z 608.39,A -85,B 0,C 180,E1 23886.294,E2 23886.294} C_VEL
LIN {X 0,Y 528.466,Z 608.4,A -85,B 0,C 180,E1 23882.854,E2 23882.854} C_VEL
LIN {X 0,Y 528.527,Z 608.403,A -85,B 0,C 180,E1 23879.588,E2 23879.588} C_VEL
LIN {X 0,Y 528.465,Z 608.401,A -85,B 0,C 180,E1 23876.257,E2 23876.257} C_VEL
LIN {X 0,Y 528.509,Z 608.401,A -85,B 0,C 180,E1 23872.878,E2 23872.878} C_VEL
LIN {X 0,Y 528.489,Z 608.392,A -85,B 0,C 180,E1 23869.565,E2 23869.565} C_VEL
LIN {X 0,Y 528.475,Z 608.393,A -85,B 0,C 180,E1 23866.148,E2 23866.148} C_VEL
LIN {X 0,Y 528.527,Z 608.404,A -85,B 0,C 180,E1 23862.899,E2 23862.899} C_VEL
LIN {X 0,Y 528.542,Z 608.72,A -85,B 0,C 180,E1 23862.26,E2 23862.26} C_VEL
LIN {X 0,Y 532.304,Z 622.848,A -85,B 0,C 180,E1 23860.17,E2 23860.17} C_VEL
LIN {X 0,Y 531.344,Z 650.255,A -85,B 0,C 180,E1 23856.7,E2 23856.7} C_VEL
LIN {X 0,Y 530.516,Z 677.132,A -85,B 0,C 180,E1 23853.35,E2 23853.35} C_VEL
LIN {X 0,Y 530.123,Z 693.133,A -85,B 0,C 180,E1 23851.405,E2 23851.405} C_VEL
LIN {X 0,Y 531.923,Z 703.547,A -85,B 0,C 180,E1 23851.158,E2 23851.158} C_VEL
LIN {X 0,Y 531.114,Z 834.934,A -85,B 0,C 180,E1 23849.292,E2 23849.292} C_VEL
LIN {X 0,Y 530.879,Z 851.869,A -85,B 0,C 180,E1 23848.833,E2 23848.833} C_VEL
LIN {X 0,Y 530.554,Z 867.017,A -85,B 0,C 180,E1 23848.218,E2 23848.218} C_VEL
LIN {X 0,Y 530.146,Z 881.74,A -85,B 0,C 180,E1 23847.406,E2 23847.406} C_VEL
LIN {X 0,Y 529.707,Z 895.517,A -85,B 0,C 180,E1 23846.429,E2 23846.429} C_VEL
LIN {X 0,Y 529.284,Z 908.179,A -85,B 0,C 180,E1 23845.287,E2 23845.287} C_VEL
LIN {X 0,Y 528.88,Z 920.126,A -85,B 0,C 180,E1 23843.945,E2 23843.945} C_VEL
LIN {X 0,Y 528.535,Z 930.32,A -85,B 0,C 180,E1 23842.5,E2 23842.5} C_VEL
LIN {X 0,Y 528.29,Z 938.932,A -85,B 0,C 180,E1 23840.962,E2 23840.962} C_VEL
LIN {X 0,Y 528.136,Z 945.66,A -85,B 0,C 180,E1 23839.418,E2 23839.418} C_VEL
LIN {X 0,Y 528.044,Z 951.314,A -85,B 0,C 180,E1 23837.645,E2 23837.645} C_VEL
LIN {X 0,Y 527.99,Z 955.118,A -85,B 0,C 180,E1 23835.86,E2 23835.86} C_VEL
LIN {X 0,Y 527.971,Z 957.06,A -85,B 0,C 180,E1 23834.062,E2 23834.062} C_VEL
LIN {X 0,Y 527.97,Z 957.296,A -85,B 0,C 180,E1 23832.248,E2 23832.248} C_VEL
LIN {X 0,Y 527.988,Z 955.662,A -85,B 0,C 180,E1 23830.416,E2 23830.416} C_VEL
LIN {X 0,Y 528.035,Z 952.423,A -85,B 0,C 180,E1 23828.681,E2 23828.681} C_VEL
LIN {X 0,Y 528.118,Z 947.352,A -85,B 0,C 180,E1 23826.944,E2 23826.944} C_VEL
LIN {X 0,Y 528.263,Z 940.593,A -85,B 0,C 180,E1 23825.273,E2 23825.273} C_VEL
LIN {X 0,Y 528.502,Z 932.403,A -85,B 0,C 180,E1 23823.724,E2 23823.724} C_VEL
LIN {X 0,Y 528.834,Z 922.352,A -85,B 0,C 180,E1 23822.233,E2 23822.233} C_VEL
LIN {X 0,Y 529.233,Z 911.309,A -85,B 0,C 180,E1 23820.918,E2 23820.918} C_VEL
LIN {X 0,Y 529.654,Z 898.822,A -85,B 0,C 180,E1 23819.733,E2 23819.733} C_VEL
LIN {X 0,Y 530.109,Z 885.142,A -85,B 0,C 180,E1 23818.696,E2 23818.696} C_VEL
LIN {X 0,Y 530.499,Z 871.558,A -85,B 0,C 180,E1 23817.893,E2 23817.893} C_VEL
LIN {X 0,Y 530.885,Z 855.552,A -85,B 0,C 180,E1 23817.184,E2 23817.184} C_VEL
LIN {X 0,Y 531.145,Z 839.645,A -85,B 0,C 180,E1 23816.699,E2 23816.699} C_VEL
LIN {X 0,Y 531.308,Z 819.589,A -85,B 0,C 180,E1 23816.352,E2 23816.352} C_VEL
LIN {X 0,Y 531.849,Z 701.244,A -85,B 0,C 180,E1 23814.678,E2 23814.678} C_VEL
LIN {X 0,Y 530.181,Z 693.101,A -85,B 0,C 180,E1 23814.457,E2 23814.457} C_VEL
LIN {X 0,Y 531.014,Z 665.328,A -85,B 0,C 180,E1 23811.032,E2 23811.032} C_VEL
LIN {X 0,Y 531.942,Z 637.815,A -85,B 0,C 180,E1 23807.562,E2 23807.562} C_VEL
LIN {X 0,Y 532.365,Z 622.626,A -85,B 0,C 180,E1 23805.614,E2 23805.614} C_VEL
LIN {X 0,Y 528.525,Z 608.525,A -85,B 0,C 180,E1 23803.439,E2 23803.439} C_VEL
LIN {X 0,Y 528.518,Z 608.396,A -85,B 0,C 180,E1 23799.988,E2 23799.988} C_VEL
LIN {X 0,Y 528.519,Z 608.4,A -85,B 0,C 180,E1 23796.444,E2 23796.444} C_VEL
LIN {X 0,Y 528.511,Z 608.398,A -85,B 0,C 180,E1 23793.015,E2 23793.015} C_VEL
LIN {X 0,Y 528.513,Z 608.397,A -85,B 0,C 180,E1 23789.589,E2 23789.589} C_VEL
LIN {X 0,Y 528.522,Z 608.399,A -85,B 0,C 180,E1 23786.155,E2 23786.155} C_VEL
LIN {X 0,Y 528.514,Z 608.397,A -85,B 0,C 180,E1 23782.702,E2 23782.702} C_VEL
LIN {X 0,Y 528.506,Z 608.396,A -85,B 0,C 180,E1 23779.334,E2 23779.334} C_VEL
LIN {X 0,Y 528.521,Z 608.403,A -85,B 0,C 180,E1 23775.921,E2 23775.921} C_VEL
LIN {X 0,Y 528.523,Z 608.395,A -85,B 0,C 180,E1 23772.455,E2 23772.455} C_VEL
LIN {X 0,Y 528.507,Z 608.399,A -85,B 0,C 180,E1 23769.034,E2 23769.034} C_VEL
LIN {X 0,Y 528.516,Z 608.396,A -85,B 0,C 180,E1 23765.646,E2 23765.646} C_VEL
LIN {X 0,Y 528.52,Z 608.394,A -85,B 0,C 180,E1 23762.169,E2 23762.169} C_VEL
LIN {X 0,Y 528.506,Z 608.401,A -85,B 0,C 180,E1 23758.699,E2 23758.699} C_VEL
LIN {X 0,Y 528.515,Z 608.391,A -85,B 0,C 180,E1 23755.334,E2 23755.334} C_VEL
LIN {X 0,Y 528.506,Z 608.393,A -85,B 0,C 180,E1 23751.952,E2 23751.952} C_VEL
LIN {X 0,Y 528.511,Z 608.401,A -85,B 0,C 180,E1 23748.432,E2 23748.432} C_VEL
LIN {X 0,Y 528.517,Z 608.393,A -85,B 0,C 180,E1 23744.979,E2 23744.979} C_VEL
LIN {X 0,Y 528.501,Z 608.39,A -85,B 0,C 180,E1 23741.582,E2 23741.582} C_VEL
LIN {X 0,Y 528.518,Z 608.399,A -85,B 0,C 180,E1 23738.119,E2 23738.119} C_VEL
LIN {X 0,Y 528.524,Z 608.397,A -85,B 0,C 180,E1 23734.688,E2 23734.688} C_VEL
LIN {X 0,Y 528.498,Z 608.4,A -85,B 0,C 180,E1 23731.279,E2 23731.279} C_VEL
LIN {X 0,Y 528.524,Z 608.398,A -85,B 0,C 180,E1 23727.887,E2 23727.887} C_VEL
LIN {X 0,Y 528.521,Z 608.394,A -85,B 0,C 180,E1 23724.361,E2 23724.361} C_VEL
LIN {X 0,Y 528.495,Z 608.401,A -85,B 0,C 180,E1 23720.95,E2 23720.95} C_VEL
LIN {X 0,Y 528.524,Z 608.403,A -85,B 0,C 180,E1 23717.517,E2 23717.517} C_VEL
LIN {X 0,Y 528.519,Z 608.396,A -85,B 0,C 180,E1 23714.037,E2 23714.037} C_VEL
LIN {X 0,Y 528.494,Z 608.402,A -85,B 0,C 180,E1 23710.603,E2 23710.603} C_VEL
LIN {X 0,Y 528.524,Z 608.404,A -85,B 0,C 180,E1 23707.208,E2 23707.208} C_VEL
LIN {X 0,Y 528.565,Z 608.68,A -85,B 0,C 180,E1 23705.067,E2 23705.067} C_VEL
LIN {X 0,Y 535.619,Z 628.831,A -85,B 0,C 180,E1 23702.903,E2 23702.903} C_VEL
LIN {X 0,Y 534.439,Z 672.306,A -85,B 0,C 180,E1 23699.548,E2 23699.548} C_VEL
LIN {X 0,Y 533.302,Z 709.709,A -85,B 0,C 180,E1 23696.678,E2 23696.678} C_VEL
LIN {X 0,Y 535.104,Z 722.369,A -85,B 0,C 180,E1 23696.388,E2 23696.388} C_VEL
LIN {X 0,Y 533.572,Z 927.53,A -85,B 0,C 180,E1 23693.455,E2 23693.455} C_VEL
LIN {X 0,Y 533.167,Z 946.957,A -85,B 0,C 180,E1 23692.973,E2 23692.973} C_VEL
LIN {X 0,Y 532.665,Z 964.796,A -85,B 0,C 180,E1 23692.34,E2 23692.34} C_VEL
LIN {X 0,Y 532.056,Z 982.788,A -85,B 0,C 180,E1 23691.497,E2 23691.497} C_VEL
LIN {X 0,Y 531.366,Z 1000.634,A -85,B 0,C 180,E1 23690.434,E2 23690.434} C_VEL
LIN {X 0,Y 530.676,Z 1017.459,A -85,B 0,C 180,E1 23689.194,E2 23689.194} C_VEL
LIN {X 0,Y 530.01,Z 1033.1,A -85,B 0,C 180,E1 23687.795,E2 23687.795} C_VEL
LIN {X 0,Y 529.448,Z 1046.684,A -85,B 0,C 180,E1 23686.343,E2 23686.343} C_VEL
LIN {X 0,Y 528.939,Z 1059.755,A -85,B 0,C 180,E1 23684.673,E2 23684.673} C_VEL
LIN {X 0,Y 528.543,Z 1071.299,A -85,B 0,C 180,E1 23682.898,E2 23682.898} C_VEL
LIN {X 0,Y 528.263,Z 1081.337,A -85,B 0,C 180,E1 23681.021,E2 23681.021} C_VEL
LIN {X 0,Y 528.077,Z 1089.433,A -85,B 0,C 180,E1 23679.151,E2 23679.151} C_VEL
LIN {X 0,Y 527.98,Z 1096.129,A -85,B 0,C 180,E1 23677.18,E2 23677.18} C_VEL
LIN {X 0,Y 527.924,Z 1101.296,A -85,B 0,C 180,E1 23675.107,E2 23675.107} C_VEL
LIN {X 0,Y 527.911,Z 1104.658,A -85,B 0,C 180,E1 23673.04,E2 23673.04} C_VEL
LIN {X 0,Y 527.909,Z 1106.304,A -85,B 0,C 180,E1 23670.976,E2 23670.976} C_VEL
LIN {X 0,Y 527.906,Z 1106.264,A -85,B 0,C 180,E1 23668.914,E2 23668.914} C_VEL
LIN {X 0,Y 527.914,Z 1104.539,A -85,B 0,C 180,E1 23666.851,E2 23666.851} C_VEL
LIN {X 0,Y 527.924,Z 1101.085,A -85,B 0,C 180,E1 23664.784,E2 23664.784} C_VEL
LIN {X 0,Y 527.983,Z 1095.818,A -85,B 0,C 180,E1 23662.71,E2 23662.71} C_VEL
LIN {X 0,Y 528.096,Z 1088.591,A -85,B 0,C 180,E1 23660.629,E2 23660.629} C_VEL
LIN {X 0,Y 528.307,Z 1079.604,A -85,B 0,C 180,E1 23658.623,E2 23658.623} C_VEL
LIN {X 0,Y 528.614,Z 1069.307,A -85,B 0,C 180,E1 23656.769,E2 23656.769} C_VEL
LIN {X 0,Y 529.03,Z 1057.322,A -85,B 0,C 180,E1 23654.993,E2 23654.993} C_VEL
LIN {X 0,Y 529.542,Z 1044.233,A -85,B 0,C 180,E1 23653.378,E2 23653.378} C_VEL
LIN {X 0,Y 530.152,Z 1029.591,A -85,B 0,C 180,E1 23651.869,E2 23651.869} C_VEL
LIN {X 0,Y 530.82,Z 1013.9,A -85,B 0,C 180,E1 23650.524,E2 23650.524} C_VEL
LIN {X 0,Y 531.5,Z 997.188,A -85,B 0,C 180,E1 23649.346,E2 23649.346} C_VEL
LIN {X 0,Y 532.162,Z 979.778,A -85,B 0,C 180,E1 23648.352,E2 23648.352} C_VEL
LIN {X 0,Y 532.744,Z 961.863,A -85,B 0,C 180,E1 23647.546,E2 23647.546} C_VEL
LIN {X 0,Y 533.234,Z 943.087,A -85,B 0,C 180,E1 23646.916,E2 23646.916} C_VEL
LIN {X 0,Y 533.612,Z 923.94,A -85,B 0,C 180,E1 23646.483,E2 23646.483} C_VEL
LIN {X 0,Y 534.943,Z 719.914,A -85,B 0,C 180,E1 23643.568,E2 23643.568} C_VEL
LIN {X 0,Y 533.255,Z 709.247,A -85,B 0,C 180,E1 23643.305,E2 23643.305} C_VEL
LIN {X 0,Y 534.654,Z 663.816,A -85,B 0,C 180,E1 23639.797,E2 23639.797} C_VEL
LIN {X 0,Y 535.673,Z 628.565,A -85,B 0,C 180,E1 23637.046,E2 23637.046} C_VEL
LIN {X 0,Y 528.565,Z 608.691,A -85,B 0,C 180,E1 23634.914,E2 23634.914} C_VEL
LIN {X 0,Y 528.511,Z 608.403,A -85,B 0,C 180,E1 23633.335,E2 23633.335} C_VEL
LIN {X 0,Y 528.504,Z 608.4,A -85,B 0,C 180,E1 23629.824,E2 23629.824} C_VEL
LIN {X 0,Y 528.516,Z 608.397,A -85,B 0,C 180,E1 23626.433,E2 23626.433} C_VEL
